LIN {X 0,Y 530.857,Z 807.028,A -85,B 0,C 180,E1 -4221.626,E2 -4221.626} C_VEL
LIN {X 0,Y 530.672,Z 814.477,A -85,B 0,C 180,E1 -4222.772,E2 -4222.772} C_VEL
LIN {X 0,Y 530.61,Z 820.462,A -85,B 0,C 180,E1 -4223.917,E2 -4223.917} C_VEL
LIN {X 0,Y 530.459,Z 825.2,A -85,B 0,C 180,E1 -4225.059,E2 -4225.059} C_VEL
LIN {X 0,Y 530.516,Z 828.828,A -85,B 0,C 180,E1 -4226.202,E2 -4226.202} C_VEL
LIN {X 0,Y 530.457,Z 830.697,A -85,B 0,C 180,E1 -4226.962,E2 -4226.962} C_VEL
LIN {X 0,Y 530.411,Z 832.131,A -85,B 0,C 180,E1 -4227.721,E2 -4227.721} C_VEL
LIN {X 0,Y 530.344,Z 833.756,A -85,B 0,C 180,E1 -4229.24,E2 -4229.24} C_VEL
LIN {X 0,Y 530.343,Z 833.996,A -85,B 0,C 180,E1 -4229.999,E2 -4229.999} C_VEL
LIN {X 0,Y 530.344,Z 833.813,A -85,B 0,C 180,E1 -4230.759,E2 -4230.759} C_VEL
LIN {X 0,Y 530.411,Z 832.265,A -85,B 0,C 180,E1 -4232.277,E2 -4232.277} C_VEL
LIN {X 0,Y 530.457,Z 830.904,A -85,B 0,C 180,E1 -4233.037,E2 -4233.037} C_VEL
LIN {X 0,Y 530.523,Z 828.033,A -85,B 0,C 180,E1 -4234.178,E2 -4234.178} C_VEL
LIN {X 0,Y 530.523,Z 824.133,A -85,B 0,C 180,E1 -4235.32,E2 -4235.32} C_VEL
LIN {X 0,Y 530.593,Z 818.515,A -85,B 0,C 180,E1 -4236.576,E2 -4236.576} C_VEL
LIN {X 0,Y 530.757,Z 811.537,A -85,B 0,C 180,E1 -4237.8,E2 -4237.8} C_VEL
LIN {X 0,Y 530.906,Z 803.362,A -85,B 0,C 180,E1 -4238.948,E2 -4238.948} C_VEL
LIN {X 0,Y 531.11,Z 794.95,A -85,B 0,C 180,E1 -4239.905,E2 -4239.905} C_VEL
LIN {X 0,Y 531.408,Z 784.646,A -85,B 0,C 180,E1 -4240.862,E2 -4240.862} C_VEL
LIN {X 0,Y 531.632,Z 773.907,A -85,B 0,C 180,E1 -4241.668,E2 -4241.668} C_VEL
LIN {X 0,Y 531.868,Z 763.248,A -85,B 0,C 180,E1 -4242.302,E2 -4242.302} C_VEL
LIN {X 0,Y 532.123,Z 750.651,A -85,B 0,C 180,E1 -4242.877,E2 -4242.877} C_VEL
LIN {X 0,Y 532.321,Z 738.262,A -85,B 0,C 180,E1 -4243.285,E2 -4243.285} C_VEL
LIN {X 0,Y 532.459,Z 725.504,A -85,B 0,C 180,E1 -4243.549,E2 -4243.549} C_VEL
LIN {X 0,Y 532.759,Z 629.988,A -85,B 0,C 180,E1 -4244.844,E2 -4244.844} C_VEL
LIN {X 0,Y 531.39,Z 621.592,A -85,B 0,C 180,E1 -4245.008,E2 -4245.008} C_VEL
LIN {X 0,Y 531.82,Z 600.643,A -85,B 0,C 180,E1 -4248.133,E2 -4248.133} C_VEL
LIN {X 0,Y 532.25,Z 580.755,A -85,B 0,C 180,E1 -4251.088,E2 -4251.088} C_VEL
LIN {X 0,Y 532.638,Z 561.67,A -85,B 0,C 180,E1 -4253.936,E2 -4253.936} C_VEL
LIN {X 0,Y 532.951,Z 545.283,A -85,B 0,C 180,E1 -4256.395,E2 -4256.395} C_VEL
LIN {X 0,Y 532.042,Z 539.407,A -85,B 0,C 180,E1 -4257.323,E2 -4257.323} C_VEL
LIN {X 0,Y 531.008,Z 534.341,A -85,B 0,C 180,E1 -4258.13,E2 -4258.13} C_VEL
LIN {X 0,Y 530.963,Z 534.35,A -85,B 0,C 180,E1 -4261.078,E2 -4261.078} C_VEL
LIN {X 0,Y 530.991,Z 534.342,A -85,B 0,C 180,E1 -4263.771,E2 -4263.771} C_VEL
LIN {X 0,Y 530.966,Z 534.341,A -85,B 0,C 180,E1 -4266.556,E2 -4266.556} C_VEL
LIN {X 0,Y 530.98,Z 534.341,A -85,B 0,C 180,E1 -4269.853,E2 -4269.853} C_VEL
LIN {X 0,Y 530.978,Z 534.339,A -85,B 0,C 180,E1 -4272.455,E2 -4272.455} C_VEL
LIN {X 0,Y 530.983,Z 534.344,A -85,B 0,C 180,E1 -4275.62,E2 -4275.62} C_VEL
LIN {X 0,Y 531.013,Z 534.336,A -85,B 0,C 180,E1 -4278.566,E2 -4278.566} C_VEL
LIN {X 0,Y 530.954,Z 534.351,A -85,B 0,C 180,E1 -4281.529,E2 -4281.529} C_VEL
LIN {X 0,Y 531.024,Z 534.342,A -85,B 0,C 180,E1 -4283.492,E2 -4283.492} C_VEL
LIN {X 0,Y 532.777,Z 540.518,A -85,B 0,C 180,E1 -4283.646,E2 -4283.646} C_VEL
LIN {X 0,Y 532.371,Z 613.502,A -85,B 0,C 180,E1 -4284.663,E2 -4284.663} C_VEL
LIN {X 0,Y 532.284,Z 626.553,A -85,B 0,C 180,E1 -4284.993,E2 -4284.993} C_VEL
LIN {X 0,Y 532.14,Z 640.049,A -85,B 0,C 180,E1 -4285.51,E2 -4285.51} C_VEL
LIN {X 0,Y 531.967,Z 650.777,A -85,B 0,C 180,E1 -4286.07,E2 -4286.07} C_VEL
LIN {X 0,Y 531.745,Z 660.944,A -85,B 0,C 180,E1 -4286.736,E2 -4286.736} C_VEL
LIN {X 0,Y 531.534,Z 670.886,A -85,B 0,C 180,E1 -4287.54,E2 -4287.54} C_VEL
LIN {X 0,Y 531.32,Z 680.523,A -85,B 0,C 180,E1 -4288.501,E2 -4288.501} C_VEL
LIN {X 0,Y 531.11,Z 689.206,A -85,B 0,C 180,E1 -4289.568,E2 -4289.568} C_VEL
LIN {X 0,Y 530.906,Z 696.438,A -85,B 0,C 180,E1 -4290.673,E2 -4290.673} C_VEL
LIN {X 0,Y 530.761,Z 703.132,A -85,B 0,C 180,E1 -4291.961,E2 -4291.961} C_VEL
LIN {X 0,Y 530.695,Z 708.251,A -85,B 0,C 180,E1 -4293.239,E2 -4293.239} C_VEL
LIN {X 0,Y 530.658,Z 711.26,A -85,B 0,C 180,E1 -4294.232,E2 -4294.232} C_VEL
LIN {X 0,Y 530.576,Z 712.968,A -85,B 0,C 180,E1 -4294.921,E2 -4294.921} C_VEL
LIN {X 0,Y 530.54,Z 714.979,A -85,B 0,C 180,E1 -4296.065,E2 -4296.065} C_VEL
LIN {X 0,Y 530.53,Z 716.161,A -85,B 0,C 180,E1 -4297.408,E2 -4297.408} C_VEL
LIN {X 0,Y 530.522,Z 716.323,A -85,B 0,C 180,E1 -4298.227,E2 -4298.227} C_VEL
LIN {X 0,Y 530.549,Z 716.011,A -85,B 0,C 180,E1 -4299.043,E2 -4299.043} C_VEL
LIN {X 0,Y 530.546,Z 714.9,A -85,B 0,C 180,E1 -4300.134,E2 -4300.134} C_VEL
LIN {X 0,Y 530.626,Z 712.421,A -85,B 0,C 180,E1 -4301.466,E2 -4301.466} C_VEL
LIN {X 0,Y 530.723,Z 708.756,A -85,B 0,C 180,E1 -4302.759,E2 -4302.759} C_VEL
LIN {X 0,Y 530.787,Z 704.588,A -85,B 0,C 180,E1 -4303.856,E2 -4303.856} C_VEL
LIN {X 0,Y 530.918,Z 698.585,A -85,B 0,C 180,E1 -4305.085,E2 -4305.085} C_VEL
LIN {X 0,Y 531.091,Z 691.628,A -85,B 0,C 180,E1 -4306.22,E2 -4306.22} C_VEL
LIN {X 0,Y 531.32,Z 682.636,A -85,B 0,C 180,E1 -4307.393,E2 -4307.393} C_VEL
LIN {X 0,Y 531.545,Z 672.652,A -85,B 0,C 180,E1 -4308.427,E2 -4308.427} C_VEL
LIN {X 0,Y 531.81,Z 662.883,A -85,B 0,C 180,E1 -4309.242,E2 -4309.242} C_VEL
LIN {X 0,Y 531.97,Z 652.92,A -85,B 0,C 180,E1 -4309.918,E2 -4309.918} C_VEL
LIN {X 0,Y 532.165,Z 641.21,A -85,B 0,C 180,E1 -4310.546,E2 -4310.546} C_VEL
LIN {X 0,Y 532.316,Z 628.322,A -85,B 0,C 180,E1 -4311.052,E2 -4311.052} C_VEL
LIN {X 0,Y 532.423,Z 615.599,A -85,B 0,C 180,E1 -4311.388,E2 -4311.388} C_VEL
LIN {X 0,Y 532.528,Z 579.636,A -85,B 0,C 180,E1 -4311.911,E2 -4311.911} C_VEL
LIN {X 0,Y 532.662,Z 539.432,A -85,B 0,C 180,E1 -4312.471,E2 -4312.471} C_VEL
LIN {X 0,Y 531.058,Z 534.338,A -85,B 0,C 180,E1 -4312.605,E2 -4312.605} C_VEL
LIN {X 0,Y 531.137,Z 534.329,A -85,B 0,C 180,E1 -4314.685,E2 -4314.685} C_VEL
LIN {X 0,Y 531.13,Z 534.321,A -85,B 0,C 180,E1 -4317.725,E2 -4317.725} C_VEL
LIN {X 0,Y 531.147,Z 534.328,A -85,B 0,C 180,E1 -4320.758,E2 -4320.758} C_VEL
LIN {X 0,Y 531.101,Z 534.329,A -85,B 0,C 180,E1 -4323.034,E2 -4323.034} C_VEL
LIN {X 0,Y 531.081,Z 534.328,A -85,B 0,C 180,E1 -4326.077,E2 -4326.077} C_VEL
LIN {X 0,Y 531.027,Z 534.336,A -85,B 0,C 180,E1 -4329.138,E2 -4329.138} C_VEL
LIN {X 0,Y 531.03,Z 534.335,A -85,B 0,C 180,E1 -4332.225,E2 -4332.225} C_VEL
LIN {X 0,Y 530.985,Z 534.338,A -85,B 0,C 180,E1 -4335.35,E2 -4335.35} C_VEL
LIN {X 0,Y 531.006,Z 534.336,A -85,B 0,C 180,E1 -4337.723,E2 -4337.723} C_VEL
LIN {X 0,Y 530.992,Z 534.344,A -85,B 0,C 180,E1 -4340.938,E2 -4340.938} C_VEL
LIN {X 0,Y 530.97,Z 534.342,A -85,B 0,C 180,E1 -4344.225,E2 -4344.225} C_VEL
LIN {X 0,Y 531.003,Z 534.344,A -85,B 0,C 180,E1 -4346.744,E2 -4346.744} C_VEL
LIN {X 0,Y 530.991,Z 534.34,A -85,B 0,C 180,E1 -4349.322,E2 -4349.322} C_VEL
LIN {X 0,Y 530.972,Z 534.341,A -85,B 0,C 180,E1 -4352.104,E2 -4352.104} C_VEL
LIN {X 0,Y 530.984,Z 534.345,A -85,B 0,C 180,E1 -4354.856,E2 -4354.856} C_VEL
LIN {X 0,Y 530.96,Z 534.341,A -85,B 0,C 180,E1 -4357.508,E2 -4357.508} C_VEL
LIN {X 0,Y 531.021,Z 534.337,A -85,B 0,C 180,E1 -4360.429,E2 -4360.429} C_VEL
LIN {X 0,Y 530.962,Z 534.344,A -85,B 0,C 180,E1 -4363.495,E2 -4363.495} C_VEL
LIN {X 0,Y 530.961,Z 534.347,A -85,B 0,C 180,E1 -4366.507,E2 -4366.507} C_VEL
LIN {X 0,Y 531.004,Z 534.338,A -85,B 0,C 180,E1 -4369.571,E2 -4369.571} C_VEL
LIN {X 0,Y 530.974,Z 534.346,A -85,B 0,C 180,E1 -4372.577,E2 -4372.577} C_VEL
LIN {X 0,Y 531.001,Z 534.341,A -85,B 0,C 180,E1 -4375.312,E2 -4375.312} C_VEL
LIN {X 0,Y 530.981,Z 534.341,A -85,B 0,C 180,E1 -4378.034,E2 -4378.034} C_VEL
LIN {X 0,Y 530.988,Z 534.347,A -85,B 0,C 180,E1 -4380.875,E2 -4380.875} C_VEL
LIN {X 0,Y 531.045,Z 534.42,A -85,B 0,C 180,E1 -4381.672,E2 -4381.672} C_VEL
LIN {X 0,Y 533.486,Z 546.142,A -85,B 0,C 180,E1 -4383.18,E2 -4383.18} C_VEL
LIN {X 0,Y 533.098,Z 569.291,A -85,B 0,C 180,E1 -4385.879,E2 -4385.879} C_VEL
LIN {X 0,Y 532.644,Z 593.969,A -85,B 0,C 180,E1 -4388.726,E2 -4388.726} C_VEL
LIN {X 0,Y 532.2,Z 621.201,A -85,B 0,C 180,E1 -4391.799,E2 -4391.799} C_VEL
LIN {X 0,Y 531.716,Z 649.824,A -85,B 0,C 180,E1 -4395.024,E2 -4395.024} C_VEL
LIN {X 0,Y 532.846,Z 659.307,A -85,B 0,C 180,E1 -4395.194,E2 -4395.194} C_VEL
LIN {X 0,Y 532.428,Z 759.985,A -85,B 0,C 180,E1 -4396.572,E2 -4396.572} C_VEL
LIN {X 0,Y 532.25,Z 773.234,A -85,B 0,C 180,E1 -4396.908,E2 -4396.908} C_VEL
LIN {X 0,Y 532.06,Z 785.381,A -85,B 0,C 180,E1 -4397.364,E2 -4397.364} C_VEL
LIN {X 0,Y 531.805,Z 797.318,A -85,B 0,C 180,E1 -4397.968,E2 -4397.968} C_VEL
LIN {X 0,Y 531.534,Z 809.205,A -85,B 0,C 180,E1 -4398.755,E2 -4398.755} C_VEL
LIN {X 0,Y 531.255,Z 819.613,A -85,B 0,C 180,E1 -4399.617,E2 -4399.617} C_VEL
LIN {X 0,Y 531.06,Z 828.121,A -85,B 0,C 180,E1 -4400.479,E2 -4400.479} C_VEL
LIN {X 0,Y 530.886,Z 835.966,A -85,B 0,C 180,E1 -4401.436,E2 -4401.436} C_VEL
LIN {X 0,Y 530.684,Z 843.627,A -85,B 0,C 180,E1 -4402.582,E2 -4402.582} C_VEL
LIN {X 0,Y 530.604,Z 850.682,A -85,B 0,C 180,E1 -4403.918,E2 -4403.918} C_VEL
LIN {X 0,Y 530.459,Z 855.375,A -85,B 0,C 180,E1 -4405.06,E2 -4405.06} C_VEL
LIN {X 0,Y 530.516,Z 858.962,A -85,B 0,C 180,E1 -4406.203,E2 -4406.203} C_VEL
LIN {X 0,Y 530.457,Z 860.811,A -85,B 0,C 180,E1 -4406.963,E2 -4406.963} C_VEL
LIN {X 0,Y 530.41,Z 862.198,A -85,B 0,C 180,E1 -4407.723,E2 -4407.723} C_VEL
LIN {X 0,Y 530.344,Z 863.787,A -85,B 0,C 180,E1 -4409.241,E2 -4409.241} C_VEL
LIN {X 0,Y 530.342,Z 864,A -85,B 0,C 180,E1 -4410.001,E2 -4410.001} C_VEL
LIN {X 0,Y 530.361,Z 863.182,A -85,B 0,C 180,E1 -4411.519,E2 -4411.519} C_VEL
LIN {X 0,Y 530.41,Z 862.193,A -85,B 0,C 180,E1 -4412.279,E2 -4412.279} C_VEL
LIN {X 0,Y 530.457,Z 860.806,A -85,B 0,C 180,E1 -4413.038,E2 -4413.038} C_VEL
LIN {X 0,Y 530.523,Z 857.893,A -85,B 0,C 180,E1 -4414.179,E2 -4414.179} C_VEL
LIN {X 0,Y 530.525,Z 853.948,A -85,B 0,C 180,E1 -4415.321,E2 -4415.321} C_VEL
LIN {X 0,Y 530.599,Z 848.261,A -85,B 0,C 180,E1 -4416.582,E2 -4416.582} C_VEL
LIN {X 0,Y 530.759,Z 841.232,A -85,B 0,C 180,E1 -4417.801,E2 -4417.801} C_VEL
LIN {X 0,Y 530.93,Z 832.988,A -85,B 0,C 180,E1 -4418.948,E2 -4418.948} C_VEL
LIN {X 0,Y 531.137,Z 824.535,A -85,B 0,C 180,E1 -4419.906,E2 -4419.906} C_VEL
LIN {X 0,Y 531.409,Z 814.086,A -85,B 0,C 180,E1 -4420.863,E2 -4420.863} C_VEL
LIN {X 0,Y 531.694,Z 803.348,A -85,B 0,C 180,E1 -4421.656,E2 -4421.656} C_VEL
LIN {X 0,Y 531.933,Z 792.398,A -85,B 0,C 180,E1 -4422.301,E2 -4422.301} C_VEL
LIN {X 0,Y 532.145,Z 780.762,A -85,B 0,C 180,E1 -4422.829,E2 -4422.829} C_VEL
LIN {X 0,Y 532.302,Z 767.334,A -85,B 0,C 180,E1 -4423.262,E2 -4423.262} C_VEL
LIN {X 0,Y 532.481,Z 754.055,A -85,B 0,C 180,E1 -4423.525,E2 -4423.525} C_VEL
LIN {X 0,Y 532.704,Z 658.004,A -85,B 0,C 180,E1 -4424.828,E2 -4424.828} C_VEL
LIN {X 0,Y 531.593,Z 650.618,A -85,B 0,C 180,E1 -4424.969,E2 -4424.969} C_VEL
LIN {X 0,Y 531.951,Z 627.9,A -85,B 0,C 180,E1 -4427.853,E2 -4427.853} C_VEL
LIN {X 0,Y 532.42,Z 604.132,A -85,B 0,C 180,E1 -4430.88,E2 -4430.88} C_VEL
LIN {X 0,Y 532.824,Z 580.756,A -85,B 0,C 180,E1 -4433.929,E2 -4433.929} C_VEL
LIN {X 0,Y 533.285,Z 560.404,A -85,B 0,C 180,E1 -4436.621,E2 -4436.621} C_VEL
LIN {X 0,Y 533.55,Z 546.301,A -85,B 0,C 180,E1 -4438.522,E2 -4438.522} C_VEL
LIN {X 0,Y 530.999,Z 534.344,A -85,B 0,C 180,E1 -4440.312,E2 -4440.312} C_VEL
LIN {X 0,Y 531.002,Z 534.34,A -85,B 0,C 180,E1 -4443.506,E2 -4443.506} C_VEL
LIN {X 0,Y 530.958,Z 534.345,A -85,B 0,C 180,E1 -4446.558,E2 -4446.558} C_VEL
LIN {X 0,Y 530.991,Z 534.341,A -85,B 0,C 180,E1 -4449.443,E2 -4449.443} C_VEL
LIN {X 0,Y 530.98,Z 534.34,A -85,B 0,C 180,E1 -4452.457,E2 -4452.457} C_VEL
LIN {X 0,Y 530.99,Z 534.34,A -85,B 0,C 180,E1 -4455.621,E2 -4455.621} C_VEL
LIN {X 0,Y 531.002,Z 534.334,A -85,B 0,C 180,E1 -4458.565,E2 -4458.565} C_VEL
LIN {X 0,Y 530.961,Z 534.344,A -85,B 0,C 180,E1 -4461.529,E2 -4461.529} C_VEL
LIN {X 0,Y 530.983,Z 534.336,A -85,B 0,C 180,E1 -4464.382,E2 -4464.382} C_VEL
LIN {X 0,Y 530.971,Z 534.347,A -85,B 0,C 180,E1 -4467.134,E2 -4467.134} C_VEL
LIN {X 0,Y 530.97,Z 534.341,A -85,B 0,C 180,E1 -4469.803,E2 -4469.803} C_VEL
LIN {X 0,Y 531.015,Z 534.334,A -85,B 0,C 180,E1 -4472.467,E2 -4472.467} C_VEL
LIN {X 0,Y 531.005,Z 534.336,A -85,B 0,C 180,E1 -4474.942,E2 -4474.942} C_VEL
LIN {X 0,Y 530.971,Z 534.34,A -85,B 0,C 180,E1 -4478.247,E2 -4478.247} C_VEL
LIN {X 0,Y 530.995,Z 534.335,A -85,B 0,C 180,E1 -4480.677,E2 -4480.677} C_VEL
LIN {X 0,Y 530.986,Z 534.335,A -85,B 0,C 180,E1 -4483.071,E2 -4483.071} C_VEL
LIN {X 0,Y 531.04,Z 534.339,A -85,B 0,C 180,E1 -4485.436,E2 -4485.436} C_VEL
LIN {X 0,Y 531.036,Z 534.327,A -85,B 0,C 180,E1 -4488.55,E2 -4488.55} C_VEL
LIN {X 0,Y 531.056,Z 534.336,A -85,B 0,C 180,E1 -4491.629,E2 -4491.629} C_VEL
LIN {X 0,Y 531.121,Z 534.32,A -85,B 0,C 180,E1 -4494.685,E2 -4494.685} C_VEL
LIN {X 0,Y 531.139,Z 534.321,A -85,B 0,C 180,E1 -4497.725,E2 -4497.725} C_VEL
LIN {X 0,Y 531.153,Z 534.317,A -85,B 0,C 180,E1 -4500.758,E2 -4500.758} C_VEL
LIN {X 0,Y 531.107,Z 534.322,A -85,B 0,C 180,E1 -4503.034,E2 -4503.034} C_VEL
LIN {X 0,Y 531.083,Z 534.328,A -85,B 0,C 180,E1 -4506.077,E2 -4506.077} C_VEL
LIN {X 0,Y 531.031,Z 534.333,A -85,B 0,C 180,E1 -4509.138,E2 -4509.138} C_VEL
LIN {X 0,Y 531.04,Z 534.329,A -85,B 0,C 180,E1 -4512.225,E2 -4512.225} C_VEL
LIN {X 0,Y 530.995,Z 534.338,A -85,B 0,C 180,E1 -4515.35,E2 -4515.35} C_VEL
LIN {X 0,Y 530.992,Z 534.334,A -85,B 0,C 180,E1 -4518.521,E2 -4518.521} C_VEL
LIN {X 0,Y 531,Z 534.335,A -85,B 0,C 180,E1 -4520.938,E2 -4520.938} C_VEL
LIN {X 0,Y 530.98,Z 534.341,A -85,B 0,C 180,E1 -4524.225,E2 -4524.225} C_VEL
LIN {X 0,Y 531.004,Z 534.335,A -85,B 0,C 180,E1 -4526.744,E2 -4526.744} C_VEL
LIN {X 0,Y 530.982,Z 534.339,A -85,B 0,C 180,E1 -4529.323,E2 -4529.323} C_VEL
LIN {X 0,Y 530.966,Z 534.348,A -85,B 0,C 180,E1 -4532.1,E2 -4532.1} C_VEL
LIN {X 0,Y 530.971,Z 534.339,A -85,B 0,C 180,E1 -4534.851,E2 -4534.851} C_VEL
LIN {X 0,Y 530.967,Z 534.342,A -85,B 0,C 180,E1 -4537.508,E2 -4537.508} C_VEL
LIN {X 0,Y 530.986,Z 534.345,A -85,B 0,C 180,E1 -4540.433,E2 -4540.433} C_VEL
LIN {X 0,Y 530.968,Z 534.338,A -85,B 0,C 180,E1 -4543.282,E2 -4543.282} C_VEL
LIN {X 0,Y 530.963,Z 534.34,A -85,B 0,C 180,E1 -4543.567,E2 -4543.567} C_VEL
LIN {X 0,Y 530.285,Z 534.433,A -85,B 0,C 180,E1 -4544.201,E2 -4544.201} C_VEL
LIN {X 0,Y 527.427,Z 534.783,A -85,B 0,C 180,E1 -4545.229,E2 -4545.229} C_VEL
LIN {X 0,Y 525.019,Z 535.088,A -85,B 0,C 180,E1 -4546.057,E2 -4546.057} C_VEL
LIN {X 0,Y 523.989,Z 535.207,A -85,B 0,C 180,E1 -4546.697,E2 -4546.697} C_VEL
LIN {X 0,Y 523.907,Z 535.215,A -85,B 0,C 180,E1 -4546.914,E2 -4546.914} C_VEL
LIN {X 0,Y 523.951,Z 535.219,A -85,B 0,C 180,E1 -4549.921,E2 -4549.921} C_VEL
LIN {X 0,Y 523.911,Z 535.222,A -85,B 0,C 180,E1 -4552.868,E2 -4552.868} C_VEL
LIN {X 0,Y 523.944,Z 535.218,A -85,B 0,C 180,E1 -4555.71,E2 -4555.71} C_VEL
LIN {X 0,Y 523.927,Z 535.226,A -85,B 0,C 180,E1 -4558.456,E2 -4558.456} C_VEL
LIN {X 0,Y 523.943,Z 535.22,A -85,B 0,C 180,E1 -4561.125,E2 -4561.125} C_VEL
LIN {X 0,Y 523.977,Z 535.252,A -85,B 0,C 180,E1 -4563.272,E2 -4563.272} C_VEL
LIN {X 0,Y 526.189,Z 546.301,A -85,B 0,C 180,E1 -4564.868,E2 -4564.868} C_VEL
LIN {X 0,Y 525.813,Z 563.993,A -85,B 0,C 180,E1 -4567.258,E2 -4567.258} C_VEL
LIN {X 0,Y 525.367,Z 586.308,A -85,B 0,C 180,E1 -4570.258,E2 -4570.258} C_VEL
LIN {X 0,Y 524.854,Z 607.393,A -85,B 0,C 180,E1 -4573.067,E2 -4573.067} C_VEL
LIN {X 0,Y 524.574,Z 620.937,A -85,B 0,C 180,E1 -4574.882,E2 -4574.882} C_VEL
LIN {X 0,Y 525.951,Z 631.321,A -85,B 0,C 180,E1 -4575.068,E2 -4575.068} C_VEL
LIN {X 0,Y 525.592,Z 730.102,A -85,B 0,C 180,E1 -4576.442,E2 -4576.442} C_VEL
LIN {X 0,Y 525.351,Z 742.698,A -85,B 0,C 180,E1 -4576.756,E2 -4576.756} C_VEL
LIN {X 0,Y 525.075,Z 755.532,A -85,B 0,C 180,E1 -4577.241,E2 -4577.241} C_VEL
LIN {X 0,Y 524.813,Z 768.516,A -85,B 0,C 180,E1 -4577.919,E2 -4577.919} C_VEL
LIN {X 0,Y 524.579,Z 779.937,A -85,B 0,C 180,E1 -4578.7,E2 -4578.7} C_VEL
LIN {X 0,Y 524.238,Z 790.15,A -85,B 0,C 180,E1 -4579.573,E2 -4579.573} C_VEL
LIN {X 0,Y 523.99,Z 799.413,A -85,B 0,C 180,E1 -4580.543,E2 -4580.543} C_VEL
LIN {X 0,Y 523.769,Z 808.366,A -85,B 0,C 180,E1 -4581.706,E2 -4581.706} C_VEL
LIN {X 0,Y 523.588,Z 815.567,A -85,B 0,C 180,E1 -4582.867,E2 -4582.867} C_VEL
LIN {X 0,Y 523.546,Z 822.19,A -85,B 0,C 180,E1 -4584.221,E2 -4584.221} C_VEL
LIN {X 0,Y 523.361,Z 826.54,A -85,B 0,C 180,E1 -4585.378,E2 -4585.378} C_VEL
LIN {X 0,Y 523.444,Z 828.829,A -85,B 0,C 180,E1 -4586.15,E2 -4586.15} C_VEL
LIN {X 0,Y 523.368,Z 830.698,A -85,B 0,C 180,E1 -4586.92,E2 -4586.92} C_VEL
LIN {X 0,Y 523.335,Z 832.132,A -85,B 0,C 180,E1 -4587.69,E2 -4587.69} C_VEL
LIN {X 0,Y 523.25,Z 833.756,A -85,B 0,C 180,E1 -4589.23,E2 -4589.23} C_VEL
LIN {X 0,Y 523.247,Z 833.997,A -85,B 0,C 180,E1 -4589.999,E2 -4589.999} C_VEL
LIN {X 0,Y 523.25,Z 833.812,A -85,B 0,C 180,E1 -4590.769,E2 -4590.769} C_VEL
LIN {X 0,Y 523.335,Z 832.264,A -85,B 0,C 180,E1 -4592.308,E2 -4592.308} C_VEL
LIN {X 0,Y 523.368,Z 830.902,A -85,B 0,C 180,E1 -4593.078,E2 -4593.078} C_VEL
LIN {X 0,Y 523.442,Z 828.031,A -85,B 0,C 180,E1 -4594.234,E2 -4594.234} C_VEL
LIN {X 0,Y 523.463,Z 824.131,A -85,B 0,C 180,E1 -4595.392,E2 -4595.392} C_VEL
LIN {X 0,Y 523.517,Z 818.972,A -85,B 0,C 180,E1 -4596.574,E2 -4596.574} C_VEL
LIN {X 0,Y 523.687,Z 811.531,A -85,B 0,C 180,E1 -4597.906,E2 -4597.906} C_VEL
LIN {X 0,Y 523.875,Z 803.356,A -85,B 0,C 180,E1 -4599.069,E2 -4599.069} C_VEL
LIN {X 0,Y 524.092,Z 794.941,A -85,B 0,C 180,E1 -4600.039,E2 -4600.039} C_VEL
LIN {X 0,Y 524.435,Z 784.667,A -85,B 0,C 180,E1 -4601.008,E2 -4601.008} C_VEL
LIN {X 0,Y 524.662,Z 774.366,A -85,B 0,C 180,E1 -4601.797,E2 -4601.797} C_VEL
LIN {X 0,Y 524.936,Z 763.313,A -85,B 0,C 180,E1 -4602.467,E2 -4602.467} C_VEL
LIN {X 0,Y 525.205,Z 750.727,A -85,B 0,C 180,E1 -4603.05,E2 -4603.05} C_VEL
LIN {X 0,Y 525.432,Z 738.334,A -85,B 0,C 180,E1 -4603.462,E2 -4603.462} C_VEL
LIN {X 0,Y 525.576,Z 725.581,A -85,B 0,C 180,E1 -4603.729,E2 -4603.729} C_VEL
LIN {X 0,Y 525.86,Z 630.572,A -85,B 0,C 180,E1 -4605.035,E2 -4605.035} C_VEL
LIN {X 0,Y 524.424,Z 621.641,A -85,B 0,C 180,E1 -4605.211,E2 -4605.211} C_VEL
LIN {X 0,Y 524.861,Z 601.08,A -85,B 0,C 180,E1 -4608.299,E2 -4608.299} C_VEL
LIN {X 0,Y 525.284,Z 581.86,A -85,B 0,C 180,E1 -4611.176,E2 -4611.176} C_VEL
LIN {X 0,Y 525.723,Z 562.71,A -85,B 0,C 180,E1 -4614.061,E2 -4614.061} C_VEL
LIN {X 0,Y 526.014,Z 545.667,A -85,B 0,C 180,E1 -4616.656,E2 -4616.656} C_VEL
LIN {X 0,Y 523.972,Z 535.219,A -85,B 0,C 180,E1 -4618.352,E2 -4618.352} C_VEL
LIN {X 0,Y 523.93,Z 535.223,A -85,B 0,C 180,E1 -4621.542,E2 -4621.542} C_VEL
LIN {X 0,Y 523.944,Z 535.218,A -85,B 0,C 180,E1 -4624.288,E2 -4624.288} C_VEL
LIN {X 0,Y 523.913,Z 535.226,A -85,B 0,C 180,E1 -4627.13,E2 -4627.13} C_VEL
LIN {X 0,Y 523.932,Z 535.217,A -85,B 0,C 180,E1 -4630.129,E2 -4630.129} C_VEL
LIN {X 0,Y 523.935,Z 535.216,A -85,B 0,C 180,E1 -4632.458,E2 -4632.458} C_VEL
LIN {X 0,Y 523.951,Z 535.221,A -85,B 0,C 180,E1 -4635.307,E2 -4635.307} C_VEL
LIN {X 0,Y 523.976,Z 535.213,A -85,B 0,C 180,E1 -4638.685,E2 -4638.685} C_VEL
LIN {X 0,Y 523.947,Z 535.221,A -85,B 0,C 180,E1 -4641.074,E2 -4641.074} C_VEL
LIN {X 0,Y 523.976,Z 535.268,A -85,B 0,C 180,E1 -4643.313,E2 -4643.313} C_VEL
LIN {X 0,Y 525.906,Z 541.232,A -85,B 0,C 180,E1 -4643.456,E2 -4643.456} C_VEL
LIN {X 0,Y 525.522,Z 614.868,A -85,B 0,C 180,E1 -4644.506,E2 -4644.506} C_VEL
LIN {X 0,Y 525.411,Z 628.218,A -85,B 0,C 180,E1 -4644.857,E2 -4644.857} C_VEL
LIN {X 0,Y 525.266,Z 640.719,A -85,B 0,C 180,E1 -4645.344,E2 -4645.344} C_VEL
LIN {X 0,Y 525.076,Z 651.455,A -85,B 0,C 180,E1 -4645.905,E2 -4645.905} C_VEL
LIN {X 0,Y 524.825,Z 662.003,A -85,B 0,C 180,E1 -4646.604,E2 -4646.604} C_VEL
LIN {X 0,Y 524.575,Z 672.723,A -85,B 0,C 180,E1 -4647.493,E2 -4647.493} C_VEL
LIN {X 0,Y 524.336,Z 682.377,A -85,B 0,C 180,E1 -4648.483,E2 -4648.483} C_VEL
LIN {X 0,Y 524.124,Z 691.021,A -85,B 0,C 180,E1 -4649.589,E2 -4649.589} C_VEL
LIN {X 0,Y 523.902,Z 697.976,A -85,B 0,C 180,E1 -4650.684,E2 -4650.684} C_VEL
LIN {X 0,Y 523.762,Z 704.572,A -85,B 0,C 180,E1 -4651.989,E2 -4651.989} C_VEL
LIN {X 0,Y 523.71,Z 709.592,A -85,B 0,C 180,E1 -4653.284,E2 -4653.284} C_VEL
LIN {X 0,Y 523.593,Z 713.226,A -85,B 0,C 180,E1 -4654.562,E2 -4654.562} C_VEL
LIN {X 0,Y 523.537,Z 715.764,A -85,B 0,C 180,E1 -4655.897,E2 -4655.897} C_VEL
LIN {X 0,Y 523.498,Z 717.012,A -85,B 0,C 180,E1 -4657.087,E2 -4657.087} C_VEL
LIN {X 0,Y 523.514,Z 717.334,A -85,B 0,C 180,E1 -4657.92,E2 -4657.92} C_VEL
LIN {X 0,Y 523.531,Z 717.191,A -85,B 0,C 180,E1 -4658.749,E2 -4658.749} C_VEL
LIN {X 0,Y 523.53,Z 716.142,A -85,B 0,C 180,E1 -4659.996,E2 -4659.996} C_VEL
LIN {X 0,Y 523.599,Z 714.112,A -85,B 0,C 180,E1 -4661.207,E2 -4661.207} C_VEL
LIN {X 0,Y 523.671,Z 711.297,A -85,B 0,C 180,E1 -4662.333,E2 -4662.333} C_VEL
LIN {X 0,Y 523.763,Z 706.82,A -85,B 0,C 180,E1 -4663.633,E2 -4663.633} C_VEL
LIN {X 0,Y 523.942,Z 700.744,A -85,B 0,C 180,E1 -4664.963,E2 -4664.963} C_VEL
LIN {X 0,Y 524.106,Z 694.572,A -85,B 0,C 180,E1 -4666.032,E2 -4666.032} C_VEL
LIN {X 0,Y 524.285,Z 687.599,A -85,B 0,C 180,E1 -4667.025,E2 -4667.025} C_VEL
LIN {X 0,Y 524.495,Z 679.311,A -85,B 0,C 180,E1 -4667.998,E2 -4667.998} C_VEL
LIN {X 0,Y 524.728,Z 668.738,A -85,B 0,C 180,E1 -4668.997,E2 -4668.997} C_VEL
LIN {X 0,Y 525.001,Z 658.347,A -85,B 0,C 180,E1 -4669.783,E2 -4669.783} C_VEL
LIN {X 0,Y 525.253,Z 646.898,A -85,B 0,C 180,E1 -4670.469,E2 -4670.469} C_VEL
LIN {X 0,Y 525.386,Z 635.089,A -85,B 0,C 180,E1 -4671.005,E2 -4671.005} C_VEL
LIN {X 0,Y 525.47,Z 621.492,A -85,B 0,C 180,E1 -4671.443,E2 -4671.443} C_VEL
LIN {X 0,Y 525.532,Z 607.858,A -85,B 0,C 180,E1 -4671.703,E2 -4671.703} C_VEL
LIN {X 0,Y 525.865,Z 540.993,A -85,B 0,C 180,E1 -4672.645,E2 -4672.645} C_VEL
LIN {X 0,Y 524.031,Z 535.214,A -85,B 0,C 180,E1 -4672.787,E2 -4672.787} C_VEL
LIN {X 0,Y 524.094,Z 535.206,A -85,B 0,C 180,E1 -4674.614,E2 -4674.614} C_VEL
LIN {X 0,Y 524.102,Z 535.197,A -85,B 0,C 180,E1 -4677.694,E2 -4677.694} C_VEL
LIN {X 0,Y 524.117,Z 535.203,A -85,B 0,C 180,E1 -4680.768,E2 -4680.768} C_VEL
LIN {X 0,Y 524.068,Z 535.204,A -85,B 0,C 180,E1 -4683.075,E2 -4683.075} C_VEL
LIN {X 0,Y 524.041,Z 535.205,A -85,B 0,C 180,E1 -4686.159,E2 -4686.159} C_VEL
LIN {X 0,Y 523.994,Z 535.211,A -85,B 0,C 180,E1 -4689.262,E2 -4689.262} C_VEL
LIN {X 0,Y 524.013,Z 535.207,A -85,B 0,C 180,E1 -4691.752,E2 -4691.752} C_VEL
LIN {X 0,Y 523.982,Z 535.213,A -85,B 0,C 180,E1 -4695.053,E2 -4695.053} C_VEL
LIN {X 0,Y 523.954,Z 535.215,A -85,B 0,C 180,E1 -4697.969,E2 -4697.969} C_VEL
LIN {X 0,Y 523.962,Z 535.217,A -85,B 0,C 180,E1 -4700.41,E2 -4700.41} C_VEL
LIN {X 0,Y 523.907,Z 535.228,A -85,B 0,C 180,E1 -4702.894,E2 -4702.894} C_VEL
LIN {X 0,Y 523.945,Z 535.216,A -85,B 0,C 180,E1 -4705.419,E2 -4705.419} C_VEL
LIN {X 0,Y 523.962,Z 535.213,A -85,B 0,C 180,E1 -4707.999,E2 -4707.999} C_VEL
LIN {X 0,Y 523.944,Z 535.224,A -85,B 0,C 180,E1 -4710.857,E2 -4710.857} C_VEL
LIN {X 0,Y 523.955,Z 535.214,A -85,B 0,C 180,E1 -4713.736,E2 -4713.736} C_VEL
LIN {X 0,Y 523.918,Z 535.223,A -85,B 0,C 180,E1 -4716.406,E2 -4716.406} C_VEL
LIN {X 0,Y 523.953,Z 535.22,A -85,B 0,C 180,E1 -4719.082,E2 -4719.082} C_VEL
LIN {X 0,Y 523.96,Z 535.215,A -85,B 0,C 180,E1 -4722.118,E2 -4722.118} C_VEL
LIN {X 0,Y 523.95,Z 535.219,A -85,B 0,C 180,E1 -4725.31,E2 -4725.31} C_VEL
LIN {X 0,Y 523.968,Z 535.22,A -85,B 0,C 180,E1 -4728.689,E2 -4728.689} C_VEL
LIN {X 0,Y 523.949,Z 535.222,A -85,B 0,C 180,E1 -4731.077,E2 -4731.077} C_VEL
LIN {X 0,Y 523.927,Z 535.22,A -85,B 0,C 180,E1 -4733.829,E2 -4733.829} C_VEL
LIN {X 0,Y 523.942,Z 535.223,A -85,B 0,C 180,E1 -4736.637,E2 -4736.637} C_VEL
LIN {X 0,Y 523.954,Z 535.221,A -85,B 0,C 180,E1 -4739.357,E2 -4739.357} C_VEL
LIN {X 0,Y 523.99,Z 535.296,A -85,B 0,C 180,E1 -4741.485,E2 -4741.485} C_VEL
LIN {X 0,Y 526.593,Z 547.998,A -85,B 0,C 180,E1 -4743.143,E2 -4743.143} C_VEL
LIN {X 0,Y 526.137,Z 571.739,A -85,B 0,C 180,E1 -4745.959,E2 -4745.959} C_VEL
LIN {X 0,Y 525.578,Z 598.018,A -85,B 0,C 180,E1 -4749.026,E2 -4749.026} C_VEL
LIN {X 0,Y 525.073,Z 624.677,A -85,B 0,C 180,E1 -4752.071,E2 -4752.071} C_VEL
LIN {X 0,Y 524.67,Z 649.011,A -85,B 0,C 180,E1 -4754.83,E2 -4754.83} C_VEL
LIN {X 0,Y 525.959,Z 659.644,A -85,B 0,C 180,E1 -4755.016,E2 -4755.016} C_VEL
LIN {X 0,Y 525.515,Z 759.406,A -85,B 0,C 180,E1 -4756.392,E2 -4756.392} C_VEL
LIN {X 0,Y 525.324,Z 772.875,A -85,B 0,C 180,E1 -4756.732,E2 -4756.732} C_VEL
LIN {X 0,Y 525.127,Z 785.226,A -85,B 0,C 180,E1 -4757.194,E2 -4757.194} C_VEL
LIN {X 0,Y 524.879,Z 796.026,A -85,B 0,C 180,E1 -4757.734,E2 -4757.734} C_VEL
LIN {X 0,Y 524.632,Z 806.604,A -85,B 0,C 180,E1 -4758.409,E2 -4758.409} C_VEL
LIN {X 0,Y 524.329,Z 817.474,A -85,B 0,C 180,E1 -4759.283,E2 -4759.283} C_VEL
LIN {X 0,Y 524.107,Z 826.34,A -85,B 0,C 180,E1 -4760.157,E2 -4760.157} C_VEL
LIN {X 0,Y 523.856,Z 834.483,A -85,B 0,C 180,E1 -4761.126,E2 -4761.126} C_VEL
LIN {X 0,Y 523.664,Z 842.471,A -85,B 0,C 180,E1 -4762.288,E2 -4762.288} C_VEL
LIN {X 0,Y 523.521,Z 848.736,A -85,B 0,C 180,E1 -4763.421,E2 -4763.421} C_VEL
LIN {X 0,Y 523.464,Z 853.951,A -85,B 0,C 180,E1 -4764.608,E2 -4764.608} C_VEL
LIN {X 0,Y 523.441,Z 857.897,A -85,B 0,C 180,E1 -4765.766,E2 -4765.766} C_VEL
LIN {X 0,Y 523.367,Z 860.811,A -85,B 0,C 180,E1 -4766.922,E2 -4766.922} C_VEL
LIN {X 0,Y 523.334,Z 862.197,A -85,B 0,C 180,E1 -4767.692,E2 -4767.692} C_VEL
LIN {X 0,Y 523.25,Z 863.786,A -85,B 0,C 180,E1 -4769.231,E2 -4769.231} C_VEL
LIN {X 0,Y 523.246,Z 864,A -85,B 0,C 180,E1 -4770.001,E2 -4770.001} C_VEL
LIN {X 0,Y 523.274,Z 863.181,A -85,B 0,C 180,E1 -4771.54,E2 -4771.54} C_VEL
LIN {X 0,Y 523.334,Z 862.192,A -85,B 0,C 180,E1 -4772.31,E2 -4772.31} C_VEL
LIN {X 0,Y 523.368,Z 860.805,A -85,B 0,C 180,E1 -4773.08,E2 -4773.08} C_VEL
LIN {X 0,Y 523.442,Z 857.893,A -85,B 0,C 180,E1 -4774.235,E2 -4774.235} C_VEL
LIN {X 0,Y 523.464,Z 853.948,A -85,B 0,C 180,E1 -4775.393,E2 -4775.393} C_VEL
LIN {X 0,Y 523.523,Z 848.726,A -85,B 0,C 180,E1 -4776.581,E2 -4776.581} C_VEL
LIN {X 0,Y 523.665,Z 842.462,A -85,B 0,C 180,E1 -4777.713,E2 -4777.713} C_VEL
LIN {X 0,Y 523.857,Z 834.473,A -85,B 0,C 180,E1 -4778.876,E2 -4778.876} C_VEL
LIN {X 0,Y 524.108,Z 826.328,A -85,B 0,C 180,E1 -4779.845,E2 -4779.845} C_VEL
LIN {X 0,Y 524.366,Z 816.392,A -85,B 0,C 180,E1 -4780.816,E2 -4780.816} C_VEL
LIN {X 0,Y 524.664,Z 805.181,A -85,B 0,C 180,E1 -4781.688,E2 -4781.688} C_VEL
LIN {X 0,Y 524.922,Z 794.118,A -85,B 0,C 180,E1 -4782.37,E2 -4782.37} C_VEL
LIN {X 0,Y 525.196,Z 781.781,A -85,B 0,C 180,E1 -4782.953,E2 -4782.953} C_VEL
LIN {X 0,Y 525.358,Z 768.777,A -85,B 0,C 180,E1 -4783.392,E2 -4783.392} C_VEL
LIN {X 0,Y 525.561,Z 754.996,A -85,B 0,C 180,E1 -4783.682,E2 -4783.682} C_VEL
LIN {X 0,Y 525.814,Z 658.698,A -85,B 0,C 180,E1 -4785.003,E2 -4785.003} C_VEL
LIN {X 0,Y 524.517,Z 649.943,A -85,B 0,C 180,E1 -4785.171,E2 -4785.171} C_VEL
LIN {X 0,Y 524.896,Z 627.276,A -85,B 0,C 180,E1 -4788.076,E2 -4788.076} C_VEL
LIN {X 0,Y 525.426,Z 604.808,A -85,B 0,C 180,E1 -4790.982,E2 -4790.982} C_VEL
LIN {X 0,Y 525.885,Z 581.556,A -85,B 0,C 180,E1 -4794.055,E2 -4794.055} C_VEL
LIN {X 0,Y 526.418,Z 560.732,A -85,B 0,C 180,E1 -4796.853,E2 -4796.853} C_VEL
LIN {X 0,Y 526.576,Z 547.156,A -85,B 0,C 180,E1 -4798.717,E2 -4798.717} C_VEL
LIN {X 0,Y 523.963,Z 535.221,A -85,B 0,C 180,E1 -4800.532,E2 -4800.532} C_VEL
LIN {X 0,Y 523.964,Z 535.215,A -85,B 0,C 180,E1 -4803.735,E2 -4803.735} C_VEL
LIN {X 0,Y 523.907,Z 535.223,A -85,B 0,C 180,E1 -4806.401,E2 -4806.401} C_VEL
LIN {X 0,Y 523.926,Z 535.227,A -85,B 0,C 180,E1 -4809.084,E2 -4809.084} C_VEL
LIN {X 0,Y 523.955,Z 535.214,A -85,B 0,C 180,E1 -4812.119,E2 -4812.119} C_VEL
LIN {X 0,Y 523.958,Z 535.22,A -85,B 0,C 180,E1 -4815.309,E2 -4815.309} C_VEL
LIN {X 0,Y 523.963,Z 535.212,A -85,B 0,C 180,E1 -4818.689,E2 -4818.689} C_VEL
LIN {X 0,Y 523.918,Z 535.218,A -85,B 0,C 180,E1 -4821.898,E2 -4821.898} C_VEL
LIN {X 0,Y 523.94,Z 535.218,A -85,B 0,C 180,E1 -4824.909,E2 -4824.909} C_VEL
LIN {X 0,Y 523.938,Z 535.216,A -85,B 0,C 180,E1 -4827.679,E2 -4827.679} C_VEL
LIN {X 0,Y 523.954,Z 535.213,A -85,B 0,C 180,E1 -4830.676,E2 -4830.676} C_VEL
LIN {X 0,Y 523.975,Z 535.212,A -85,B 0,C 180,E1 -4833.728,E2 -4833.728} C_VEL
LIN {X 0,Y 523.926,Z 535.214,A -85,B 0,C 180,E1 -4836.27,E2 -4836.27} C_VEL
LIN {X 0,Y 523.946,Z 535.216,A -85,B 0,C 180,E1 -4838.767,E2 -4838.767} C_VEL
LIN {X 0,Y 523.952,Z 535.218,A -85,B 0,C 180,E1 -4841.221,E2 -4841.221} C_VEL
LIN {X 0,Y 523.937,Z 535.222,A -85,B 0,C 180,E1 -4843.639,E2 -4843.639} C_VEL
LIN {X 0,Y 523.944,Z 535.217,A -85,B 0,C 180,E1 -4846.028,E2 -4846.028} C_VEL
LIN {X 0,Y 524.012,Z 535.202,A -85,B 0,C 180,E1 -4848.394,E2 -4848.394} C_VEL
LIN {X 0,Y 524.004,Z 535.212,A -85,B 0,C 180,E1 -4851.516,E2 -4851.516} C_VEL
LIN {X 0,Y 524.083,Z 535.197,A -85,B 0,C 180,E1 -4854.614,E2 -4854.614} C_VEL
LIN {X 0,Y 524.111,Z 535.196,A -85,B 0,C 180,E1 -4857.695,E2 -4857.695} C_VEL
LIN {X 0,Y 524.123,Z 535.193,A -85,B 0,C 180,E1 -4860.768,E2 -4860.768} C_VEL
LIN {X 0,Y 524.073,Z 535.199,A -85,B 0,C 180,E1 -4863.075,E2 -4863.075} C_VEL
LIN {X 0,Y 524.046,Z 535.204,A -85,B 0,C 180,E1 -4866.159,E2 -4866.159} C_VEL
LIN {X 0,Y 523.999,Z 535.21,A -85,B 0,C 180,E1 -4869.262,E2 -4869.262} C_VEL
LIN {X 0,Y 524.002,Z 535.211,A -85,B 0,C 180,E1 -4871.74,E2 -4871.74} C_VEL
LIN {X 0,Y 523.992,Z 535.209,A -85,B 0,C 180,E1 -4875.052,E2 -4875.052} C_VEL
LIN {X 0,Y 523.964,Z 535.216,A -85,B 0,C 180,E1 -4877.969,E2 -4877.969} C_VEL
LIN {X 0,Y 523.972,Z 535.213,A -85,B 0,C 180,E1 -4880.41,E2 -4880.41} C_VEL
LIN {X 0,Y 523.917,Z 535.218,A -85,B 0,C 180,E1 -4882.893,E2 -4882.893} C_VEL
LIN {X 0,Y 523.953,Z 535.211,A -85,B 0,C 180,E1 -4885.419,E2 -4885.419} C_VEL
LIN {X 0,Y 523.97,Z 535.22,A -85,B 0,C 180,E1 -4887.999,E2 -4887.999} C_VEL
LIN {X 0,Y 523.945,Z 535.212,A -85,B 0,C 180,E1 -4890.855,E2 -4890.855} C_VEL
LIN {X 0,Y 523.96,Z 535.218,A -85,B 0,C 180,E1 -4893.735,E2 -4893.735} C_VEL
LIN {X 0,Y 523.904,Z 535.227,A -85,B 0,C 180,E1 -4896.402,E2 -4896.402} C_VEL
LIN {X 0,Y 523.924,Z 535.217,A -85,B 0,C 180,E1 -4899.085,E2 -4899.085} C_VEL
LIN {X 0,Y 523.958,Z 535.223,A -85,B 0,C 180,E1 -4902.119,E2 -4902.119} C_VEL
LIN {X 0,Y 523.946,Z 535.215,A -85,B 0,C 180,E1 -4905.31,E2 -4905.31} C_VEL
LIN {X 0,Y 523.907,Z 535.215,A -85,B 0,C 180,E1 -4906.914,E2 -4906.914} C_VEL
LIN {X 0,Y 523.248,Z 535.297,A -85,B 0,C 180,E1 -4907.555,E2 -4907.555} C_VEL
LIN {X 0,Y 520.412,Z 535.663,A -85,B 0,C 180,E1 -4908.597,E2 -4908.597} C_VEL
LIN {X 0,Y 518.008,Z 535.97,A -85,B 0,C 180,E1 -4909.436,E2 -4909.436} C_VEL
LIN {X 0,Y 516.971,Z 536.096,A -85,B 0,C 180,E1 -4910.084,E2 -4910.084} C_VEL
LIN {X 0,Y 516.883,Z 536.103,A -85,B 0,C 180,E1 -4910.303,E2 -4910.303} C_VEL
LIN {X 0,Y 516.881,Z 536.096,A -85,B 0,C 180,E1 -4913.343,E2 -4913.343} C_VEL
LIN {X 0,Y 516.914,Z 536.098,A -85,B 0,C 180,E1 -4916.121,E2 -4916.121} C_VEL
LIN {X 0,Y 516.895,Z 536.101,A -85,B 0,C 180,E1 -4918.936,E2 -4918.936} C_VEL
LIN {X 0,Y 516.923,Z 536.094,A -85,B 0,C 180,E1 -4921.585,E2 -4921.585} C_VEL
LIN {X 0,Y 516.945,Z 536.202,A -85,B 0,C 180,E1 -4923.07,E2 -4923.07} C_VEL
LIN {X 0,Y 519.32,Z 547.734,A -85,B 0,C 180,E1 -4924.757,E2 -4924.757} C_VEL
LIN {X 0,Y 518.902,Z 565.545,A -85,B 0,C 180,E1 -4927.19,E2 -4927.19} C_VEL
LIN {X 0,Y 518.349,Z 589.145,A -85,B 0,C 180,E1 -4930.392,E2 -4930.392} C_VEL
LIN {X 0,Y 517.838,Z 611.858,A -85,B 0,C 180,E1 -4933.44,E2 -4933.44} C_VEL
LIN {X 0,Y 517.67,Z 621.338,A -85,B 0,C 180,E1 -4934.68,E2 -4934.68} C_VEL
LIN {X 0,Y 519.094,Z 631.643,A -85,B 0,C 180,E1 -4934.869,E2 -4934.869} C_VEL
LIN {X 0,Y 518.707,Z 730.232,A -85,B 0,C 180,E1 -4936.259,E2 -4936.259} C_VEL
LIN {X 0,Y 518.468,Z 742.855,A -85,B 0,C 180,E1 -4936.577,E2 -4936.577} C_VEL
LIN {X 0,Y 518.17,Z 755.705,A -85,B 0,C 180,E1 -4937.068,E2 -4937.068} C_VEL
LIN {X 0,Y 517.878,Z 768.47,A -85,B 0,C 180,E1 -4937.741,E2 -4937.741} C_VEL
LIN {X 0,Y 517.612,Z 780.123,A -85,B 0,C 180,E1 -4938.546,E2 -4938.546} C_VEL
LIN {X 0,Y 517.243,Z 790.339,A -85,B 0,C 180,E1 -4939.43,E2 -4939.43} C_VEL
LIN {X 0,Y 516.975,Z 799.586,A -85,B 0,C 180,E1 -4940.413,E2 -4940.413} C_VEL
LIN {X 0,Y 516.725,Z 808.503,A -85,B 0,C 180,E1 -4941.592,E2 -4941.592} C_VEL
LIN {X 0,Y 516.515,Z 815.671,A -85,B 0,C 180,E1 -4942.769,E2 -4942.769} C_VEL
LIN {X 0,Y 516.436,Z 820.542,A -85,B 0,C 180,E1 -4943.749,E2 -4943.749} C_VEL
LIN {X 0,Y 516.314,Z 825.255,A -85,B 0,C 180,E1 -4944.923,E2 -4944.923} C_VEL
LIN {X 0,Y 516.373,Z 828.859,A -85,B 0,C 180,E1 -4946.097,E2 -4946.097} C_VEL
LIN {X 0,Y 516.283,Z 830.718,A -85,B 0,C 180,E1 -4946.878,E2 -4946.878} C_VEL
LIN {X 0,Y 516.261,Z 832.143,A -85,B 0,C 180,E1 -4947.659,E2 -4947.659} C_VEL
LIN {X 0,Y 516.16,Z 833.759,A -85,B 0,C 180,E1 -4949.219,E2 -4949.219} C_VEL
LIN {X 0,Y 516.155,Z 833.998,A -85,B 0,C 180,E1 -4949.999,E2 -4949.999} C_VEL
LIN {X 0,Y 516.16,Z 833.814,A -85,B 0,C 180,E1 -4950.779,E2 -4950.779} C_VEL
LIN {X 0,Y 516.261,Z 832.272,A -85,B 0,C 180,E1 -4952.34,E2 -4952.34} C_VEL
LIN {X 0,Y 516.283,Z 830.918,A -85,B 0,C 180,E1 -4953.121,E2 -4953.121} C_VEL
LIN {X 0,Y 516.344,Z 828.064,A -85,B 0,C 180,E1 -4954.293,E2 -4954.293} C_VEL
LIN {X 0,Y 516.4,Z 824.186,A -85,B 0,C 180,E1 -4955.466,E2 -4955.466} C_VEL
LIN {X 0,Y 516.479,Z 818.386,A -85,B 0,C 180,E1 -4956.798,E2 -4956.798} C_VEL
LIN {X 0,Y 516.639,Z 811.646,A -85,B 0,C 180,E1 -4958.014,E2 -4958.014} C_VEL
LIN {X 0,Y 516.853,Z 803.504,A -85,B 0,C 180,E1 -4959.193,E2 -4959.193} C_VEL
LIN {X 0,Y 517.087,Z 795.118,A -85,B 0,C 180,E1 -4960.176,E2 -4960.176} C_VEL
LIN {X 0,Y 517.461,Z 784.84,A -85,B 0,C 180,E1 -4961.159,E2 -4961.159} C_VEL
LIN {X 0,Y 517.746,Z 774.253,A -85,B 0,C 180,E1 -4961.976,E2 -4961.976} C_VEL
LIN {X 0,Y 518.002,Z 763.467,A -85,B 0,C 180,E1 -4962.636,E2 -4962.636} C_VEL
LIN {X 0,Y 518.314,Z 750.865,A -85,B 0,C 180,E1 -4963.226,E2 -4963.226} C_VEL
LIN {X 0,Y 518.552,Z 738.438,A -85,B 0,C 180,E1 -4963.644,E2 -4963.644} C_VEL
LIN {X 0,Y 518.697,Z 725.614,A -85,B 0,C 180,E1 -4963.915,E2 -4963.915} C_VEL
LIN {X 0,Y 519.019,Z 631.443,A -85,B 0,C 180,E1 -4965.226,E2 -4965.226} C_VEL
LIN {X 0,Y 517.453,Z 621.537,A -85,B 0,C 180,E1 -4965.437,E2 -4965.437} C_VEL
LIN {X 0,Y 517.889,Z 602.176,A -85,B 0,C 180,E1 -4968.37,E2 -4968.37} C_VEL
LIN {X 0,Y 518.338,Z 582.971,A -85,B 0,C 180,E1 -4971.265,E2 -4971.265} C_VEL
LIN {X 0,Y 518.818,Z 563.789,A -85,B 0,C 180,E1 -4974.189,E2 -4974.189} C_VEL
LIN {X 0,Y 519.161,Z 547.558,A -85,B 0,C 180,E1 -4976.688,E2 -4976.688} C_VEL
LIN {X 0,Y 516.923,Z 536.098,A -85,B 0,C 180,E1 -4978.552,E2 -4978.552} C_VEL
LIN {X 0,Y 516.889,Z 536.102,A -85,B 0,C 180,E1 -4981.108,E2 -4981.108} C_VEL
LIN {X 0,Y 516.912,Z 536.095,A -85,B 0,C 180,E1 -4983.966,E2 -4983.966} C_VEL
LIN {X 0,Y 516.881,Z 536.097,A -85,B 0,C 180,E1 -4986.744,E2 -4986.744} C_VEL
LIN {X 0,Y 516.878,Z 536.099,A -85,B 0,C 180,E1 -4989.72,E2 -4989.72} C_VEL
LIN {X 0,Y 516.901,Z 536.094,A -85,B 0,C 180,E1 -4992.76,E2 -4992.76} C_VEL
LIN {X 0,Y 516.917,Z 536.092,A -85,B 0,C 180,E1 -4995.009,E2 -4995.009} C_VEL
LIN {X 0,Y 516.923,Z 536.091,A -85,B 0,C 180,E1 -4998.396,E2 -4998.396} C_VEL
LIN {X 0,Y 516.9,Z 536.101,A -85,B 0,C 180,E1 -5001.286,E2 -5001.286} C_VEL
LIN {X 0,Y 516.908,Z 536.099,A -85,B 0,C 180,E1 -5003.105,E2 -5003.105} C_VEL
LIN {X 0,Y 518.995,Z 542.487,A -85,B 0,C 180,E1 -5003.268,E2 -5003.268} C_VEL
LIN {X 0,Y 518.627,Z 616.208,A -85,B 0,C 180,E1 -5004.344,E2 -5004.344} C_VEL
LIN {X 0,Y 518.53,Z 628.771,A -85,B 0,C 180,E1 -5004.679,E2 -5004.679} C_VEL
LIN {X 0,Y 518.378,Z 641.334,A -85,B 0,C 180,E1 -5005.172,E2 -5005.172} C_VEL
LIN {X 0,Y 518.148,Z 653.583,A -85,B 0,C 180,E1 -5005.829,E2 -5005.829} C_VEL
LIN {X 0,Y 517.9,Z 664.011,A -85,B 0,C 180,E1 -5006.544,E2 -5006.544} C_VEL
LIN {X 0,Y 517.653,Z 674.21,A -85,B 0,C 180,E1 -5007.413,E2 -5007.413} C_VEL
LIN {X 0,Y 517.368,Z 684.18,A -85,B 0,C 180,E1 -5008.467,E2 -5008.467} C_VEL
LIN {X 0,Y 517.128,Z 692.664,A -85,B 0,C 180,E1 -5009.586,E2 -5009.586} C_VEL
LIN {X 0,Y 516.91,Z 699.506,A -85,B 0,C 180,E1 -5010.695,E2 -5010.695} C_VEL
LIN {X 0,Y 516.771,Z 705.482,A -85,B 0,C 180,E1 -5011.899,E2 -5011.899} C_VEL
LIN {X 0,Y 516.687,Z 710.888,A -85,B 0,C 180,E1 -5013.329,E2 -5013.329} C_VEL
LIN {X 0,Y 516.613,Z 713.401,A -85,B 0,C 180,E1 -5014.194,E2 -5014.194} C_VEL
LIN {X 0,Y 516.553,Z 715.364,A -85,B 0,C 180,E1 -5015.053,E2 -5015.053} C_VEL
LIN {X 0,Y 516.517,Z 716.805,A -85,B 0,C 180,E1 -5015.908,E2 -5015.908} C_VEL
LIN {X 0,Y 516.492,Z 717.791,A -85,B 0,C 180,E1 -5016.758,E2 -5016.758} C_VEL
LIN {X 0,Y 516.504,Z 718.288,A -85,B 0,C 180,E1 -5017.705,E2 -5017.705} C_VEL
LIN {X 0,Y 516.529,Z 717.909,A -85,B 0,C 180,E1 -5019.282,E2 -5019.282} C_VEL
LIN {X 0,Y 516.514,Z 717.035,A -85,B 0,C 180,E1 -5020.113,E2 -5020.113} C_VEL
LIN {X 0,Y 516.555,Z 715.728,A -85,B 0,C 180,E1 -5020.941,E2 -5020.941} C_VEL
LIN {X 0,Y 516.673,Z 712.832,A -85,B 0,C 180,E1 -5022.202,E2 -5022.202} C_VEL
LIN {X 0,Y 516.734,Z 708.995,A -85,B 0,C 180,E1 -5023.404,E2 -5023.404} C_VEL
LIN {X 0,Y 516.908,Z 703.977,A -85,B 0,C 180,E1 -5024.607,E2 -5024.607} C_VEL
LIN {X 0,Y 517.102,Z 697.406,A -85,B 0,C 180,E1 -5025.839,E2 -5025.839} C_VEL
LIN {X 0,Y 517.333,Z 689.305,A -85,B 0,C 180,E1 -5027.047,E2 -5027.047} C_VEL
LIN {X 0,Y 517.557,Z 680.789,A -85,B 0,C 180,E1 -5028.074,E2 -5028.074} C_VEL
LIN {X 0,Y 517.784,Z 670.819,A -85,B 0,C 180,E1 -5029.046,E2 -5029.046} C_VEL
LIN {X 0,Y 518.11,Z 659.216,A -85,B 0,C 180,E1 -5029.942,E2 -5029.942} C_VEL
LIN {X 0,Y 518.371,Z 647.693,A -85,B 0,C 180,E1 -5030.637,E2 -5030.637} C_VEL
LIN {X 0,Y 518.528,Z 635.771,A -85,B 0,C 180,E1 -5031.18,E2 -5031.18} C_VEL
LIN {X 0,Y 518.597,Z 622.622,A -85,B 0,C 180,E1 -5031.608,E2 -5031.608} C_VEL
LIN {X 0,Y 518.67,Z 609.626,A -85,B 0,C 180,E1 -5031.862,E2 -5031.862} C_VEL
LIN {X 0,Y 518.953,Z 542.348,A -85,B 0,C 180,E1 -5032.832,E2 -5032.832} C_VEL
LIN {X 0,Y 516.995,Z 536.089,A -85,B 0,C 180,E1 -5032.998,E2 -5032.998} C_VEL
LIN {X 0,Y 516.934,Z 536.092,A -85,B 0,C 180,E1 -5035.321,E2 -5035.321} C_VEL
LIN {X 0,Y 517.075,Z 536.073,A -85,B 0,C 180,E1 -5037.663,E2 -5037.663} C_VEL
LIN {X 0,Y 517.087,Z 536.079,A -85,B 0,C 180,E1 -5040.779,E2 -5040.779} C_VEL
LIN {X 0,Y 517.008,Z 536.083,A -85,B 0,C 180,E1 -5043.117,E2 -5043.117} C_VEL
LIN {X 0,Y 517.004,Z 536.083,A -85,B 0,C 180,E1 -5046.243,E2 -5046.243} C_VEL
LIN {X 0,Y 516.948,Z 536.087,A -85,B 0,C 180,E1 -5049.389,E2 -5049.389} C_VEL
LIN {X 0,Y 516.972,Z 536.085,A -85,B 0,C 180,E1 -5051.824,E2 -5051.824} C_VEL
LIN {X 0,Y 516.935,Z 536.09,A -85,B 0,C 180,E1 -5055.148,E2 -5055.148} C_VEL
LIN {X 0,Y 516.915,Z 536.093,A -85,B 0,C 180,E1 -5058.223,E2 -5058.223} C_VEL
LIN {X 0,Y 516.903,Z 536.101,A -85,B 0,C 180,E1 -5060.702,E2 -5060.702} C_VEL
LIN {X 0,Y 516.901,Z 536.094,A -85,B 0,C 180,E1 -5064.073,E2 -5064.073} C_VEL
LIN {X 0,Y 516.92,Z 536.097,A -85,B 0,C 180,E1 -5066.658,E2 -5066.658} C_VEL
LIN {X 0,Y 516.916,Z 536.092,A -85,B 0,C 180,E1 -5069.527,E2 -5069.527} C_VEL
LIN {X 0,Y 516.893,Z 536.1,A -85,B 0,C 180,E1 -5072.545,E2 -5072.545} C_VEL
LIN {X 0,Y 516.876,Z 536.099,A -85,B 0,C 180,E1 -5075.334,E2 -5075.334} C_VEL
LIN {X 0,Y 516.875,Z 536.095,A -85,B 0,C 180,E1 -5077.944,E2 -5077.944} C_VEL
LIN {X 0,Y 516.902,Z 536.099,A -85,B 0,C 180,E1 -5080.74,E2 -5080.74} C_VEL
LIN {X 0,Y 516.877,Z 536.097,A -85,B 0,C 180,E1 -5083.904,E2 -5083.904} C_VEL
LIN {X 0,Y 516.876,Z 536.098,A -85,B 0,C 180,E1 -5086.108,E2 -5086.108} C_VEL
LIN {X 0,Y 516.899,Z 536.098,A -85,B 0,C 180,E1 -5089.261,E2 -5089.261} C_VEL
LIN {X 0,Y 516.881,Z 536.097,A -85,B 0,C 180,E1 -5092.057,E2 -5092.057} C_VEL
LIN {X 0,Y 516.893,Z 536.101,A -85,B 0,C 180,E1 -5095.177,E2 -5095.177} C_VEL
LIN {X 0,Y 516.88,Z 536.098,A -85,B 0,C 180,E1 -5097.977,E2 -5097.977} C_VEL
LIN {X 0,Y 516.939,Z 536.141,A -85,B 0,C 180,E1 -5101.282,E2 -5101.282} C_VEL
LIN {X 0,Y 519.636,Z 548.741,A -85,B 0,C 180,E1 -5102.968,E2 -5102.968} C_VEL
LIN {X 0,Y 519.232,Z 568.874,A -85,B 0,C 180,E1 -5105.405,E2 -5105.405} C_VEL
LIN {X 0,Y 518.742,Z 591.806,A -85,B 0,C 180,E1 -5108.127,E2 -5108.127} C_VEL
LIN {X 0,Y 518.206,Z 618.434,A -85,B 0,C 180,E1 -5111.231,E2 -5111.231} C_VEL
LIN {X 0,Y 517.636,Z 647.918,A -85,B 0,C 180,E1 -5114.627,E2 -5114.627} C_VEL
LIN {X 0,Y 519.073,Z 661.058,A -85,B 0,C 180,E1 -5114.853,E2 -5114.853} C_VEL
LIN {X 0,Y 518.617,Z 757.64,A -85,B 0,C 180,E1 -5116.208,E2 -5116.208} C_VEL
LIN {X 0,Y 518.323,Z 771.36,A -85,B 0,C 180,E1 -5116.549,E2 -5116.549} C_VEL
LIN {X 0,Y 518.108,Z 784.963,A -85,B 0,C 180,E1 -5117.067,E2 -5117.067} C_VEL
LIN {X 0,Y 517.804,Z 797.423,A -85,B 0,C 180,E1 -5117.721,E2 -5117.721} C_VEL
LIN {X 0,Y 517.494,Z 809.572,A -85,B 0,C 180,E1 -5118.545,E2 -5118.545} C_VEL
LIN {X 0,Y 517.178,Z 819.98,A -85,B 0,C 180,E1 -5119.43,E2 -5119.43} C_VEL
LIN {X 0,Y 516.938,Z 829.383,A -85,B 0,C 180,E1 -5120.414,E2 -5120.414} C_VEL
LIN {X 0,Y 516.716,Z 838.526,A -85,B 0,C 180,E1 -5121.593,E2 -5121.593} C_VEL
LIN {X 0,Y 516.509,Z 845.812,A -85,B 0,C 180,E1 -5122.77,E2 -5122.77} C_VEL
LIN {X 0,Y 516.426,Z 850.679,A -85,B 0,C 180,E1 -5123.75,E2 -5123.75} C_VEL
LIN {X 0,Y 516.313,Z 855.374,A -85,B 0,C 180,E1 -5124.925,E2 -5124.925} C_VEL
LIN {X 0,Y 516.355,Z 858.962,A -85,B 0,C 180,E1 -5126.098,E2 -5126.098} C_VEL
LIN {X 0,Y 516.282,Z 860.811,A -85,B 0,C 180,E1 -5126.879,E2 -5126.879} C_VEL
LIN {X 0,Y 516.26,Z 862.196,A -85,B 0,C 180,E1 -5127.66,E2 -5127.66} C_VEL
LIN {X 0,Y 516.16,Z 863.786,A -85,B 0,C 180,E1 -5129.221,E2 -5129.221} C_VEL
LIN {X 0,Y 516.154,Z 864,A -85,B 0,C 180,E1 -5130.001,E2 -5130.001} C_VEL
LIN {X 0,Y 516.192,Z 863.181,A -85,B 0,C 180,E1 -5131.561,E2 -5131.561} C_VEL
LIN {X 0,Y 516.26,Z 862.192,A -85,B 0,C 180,E1 -5132.341,E2 -5132.341} C_VEL
LIN {X 0,Y 516.283,Z 860.805,A -85,B 0,C 180,E1 -5133.122,E2 -5133.122} C_VEL
LIN {X 0,Y 516.344,Z 857.892,A -85,B 0,C 180,E1 -5134.294,E2 -5134.294} C_VEL
LIN {X 0,Y 516.405,Z 853.948,A -85,B 0,C 180,E1 -5135.467,E2 -5135.467} C_VEL
LIN {X 0,Y 516.487,Z 848.013,A -85,B 0,C 180,E1 -5136.808,E2 -5136.808} C_VEL
LIN {X 0,Y 516.641,Z 841.12,A -85,B 0,C 180,E1 -5138.016,E2 -5138.016} C_VEL
LIN {X 0,Y 516.845,Z 832.68,A -85,B 0,C 180,E1 -5139.194,E2 -5139.194} C_VEL
LIN {X 0,Y 517.067,Z 824.014,A -85,B 0,C 180,E1 -5140.178,E2 -5140.178} C_VEL
LIN {X 0,Y 517.417,Z 813.35,A -85,B 0,C 180,E1 -5141.161,E2 -5141.161} C_VEL
LIN {X 0,Y 517.669,Z 801.623,A -85,B 0,C 180,E1 -5142.029,E2 -5142.029} C_VEL
LIN {X 0,Y 518,Z 789.265,A -85,B 0,C 180,E1 -5142.737,E2 -5142.737} C_VEL
LIN {X 0,Y 518.282,Z 776.716,A -85,B 0,C 180,E1 -5143.278,E2 -5143.278} C_VEL
LIN {X 0,Y 518.516,Z 763.765,A -85,B 0,C 180,E1 -5143.672,E2 -5143.672} C_VEL
LIN {X 0,Y 518.651,Z 748.396,A -85,B 0,C 180,E1 -5143.943,E2 -5143.943} C_VEL
LIN {X 0,Y 519.006,Z 659.922,A -85,B 0,C 180,E1 -5145.17,E2 -5145.17} C_VEL
LIN {X 0,Y 517.506,Z 649.013,A -85,B 0,C 180,E1 -5145.388,E2 -5145.388} C_VEL
LIN {X 0,Y 517.959,Z 624.734,A -85,B 0,C 180,E1 -5148.554,E2 -5148.554} C_VEL
LIN {X 0,Y 518.464,Z 604.178,A -85,B 0,C 180,E1 -5151.261,E2 -5151.261} C_VEL
LIN {X 0,Y 518.984,Z 580.795,A -85,B 0,C 180,E1 -5154.395,E2 -5154.395} C_VEL
LIN {X 0,Y 519.574,Z 558.963,A -85,B 0,C 180,E1 -5157.381,E2 -5157.381} C_VEL
LIN {X 0,Y 519.76,Z 549.106,A -85,B 0,C 180,E1 -5158.755,E2 -5158.755} C_VEL
LIN {X 0,Y 516.908,Z 536.1,A -85,B 0,C 180,E1 -5160.757,E2 -5160.757} C_VEL
LIN {X 0,Y 516.914,Z 536.093,A -85,B 0,C 180,E1 -5163.967,E2 -5163.967} C_VEL
LIN {X 0,Y 516.879,Z 536.102,A -85,B 0,C 180,E1 -5166.746,E2 -5166.746} C_VEL
LIN {X 0,Y 516.885,Z 536.096,A -85,B 0,C 180,E1 -5169.721,E2 -5169.721} C_VEL
LIN {X 0,Y 516.915,Z 536.092,A -85,B 0,C 180,E1 -5171.775,E2 -5171.775} C_VEL
LIN {X 0,Y 516.925,Z 536.094,A -85,B 0,C 180,E1 -5175.01,E2 -5175.01} C_VEL
LIN {X 0,Y 516.919,Z 536.087,A -85,B 0,C 180,E1 -5178.398,E2 -5178.398} C_VEL
LIN {X 0,Y 516.885,Z 536.102,A -85,B 0,C 180,E1 -5181.284,E2 -5181.284} C_VEL
LIN {X 0,Y 516.892,Z 536.091,A -85,B 0,C 180,E1 -5184.221,E2 -5184.221} C_VEL
LIN {X 0,Y 516.897,Z 536.099,A -85,B 0,C 180,E1 -5187.053,E2 -5187.053} C_VEL
LIN {X 0,Y 516.892,Z 536.094,A -85,B 0,C 180,E1 -5189.796,E2 -5189.796} C_VEL
LIN {X 0,Y 516.928,Z 536.089,A -85,B 0,C 180,E1 -5192.467,E2 -5192.467} C_VEL
LIN {X 0,Y 516.909,Z 536.093,A -85,B 0,C 180,E1 -5195.072,E2 -5195.072} C_VEL
LIN {X 0,Y 516.885,Z 536.094,A -85,B 0,C 180,E1 -5198.462,E2 -5198.462} C_VEL
LIN {X 0,Y 516.903,Z 536.093,A -85,B 0,C 180,E1 -5200.955,E2 -5200.955} C_VEL
LIN {X 0,Y 516.914,Z 536.092,A -85,B 0,C 180,E1 -5203.41,E2 -5203.41} C_VEL
LIN {X 0,Y 516.905,Z 536.096,A -85,B 0,C 180,E1 -5205.834,E2 -5205.834} C_VEL
LIN {X 0,Y 516.951,Z 536.084,A -85,B 0,C 180,E1 -5209.028,E2 -5209.028} C_VEL
LIN {X 0,Y 516.978,Z 536.084,A -85,B 0,C 180,E1 -5212.187,E2 -5212.187} C_VEL
LIN {X 0,Y 517.03,Z 536.076,A -85,B 0,C 180,E1 -5214.54,E2 -5214.54} C_VEL
LIN {X 0,Y 517.083,Z 536.07,A -85,B 0,C 180,E1 -5217.663,E2 -5217.663} C_VEL
LIN {X 0,Y 517.093,Z 536.068,A -85,B 0,C 180,E1 -5220.779,E2 -5220.779} C_VEL
LIN {X 0,Y 517.014,Z 536.078,A -85,B 0,C 180,E1 -5223.117,E2 -5223.117} C_VEL
LIN {X 0,Y 517.01,Z 536.079,A -85,B 0,C 180,E1 -5226.243,E2 -5226.243} C_VEL
LIN {X 0,Y 516.954,Z 536.089,A -85,B 0,C 180,E1 -5229.389,E2 -5229.389} C_VEL
LIN {X 0,Y 516.952,Z 536.088,A -85,B 0,C 180,E1 -5231.807,E2 -5231.807} C_VEL
LIN {X 0,Y 516.944,Z 536.087,A -85,B 0,C 180,E1 -5235.147,E2 -5235.147} C_VEL
LIN {X 0,Y 516.926,Z 536.088,A -85,B 0,C 180,E1 -5238.222,E2 -5238.222} C_VEL
LIN {X 0,Y 516.912,Z 536.09,A -85,B 0,C 180,E1 -5240.702,E2 -5240.702} C_VEL
LIN {X 0,Y 516.912,Z 536.095,A -85,B 0,C 180,E1 -5244.072,E2 -5244.072} C_VEL
LIN {X 0,Y 516.926,Z 536.09,A -85,B 0,C 180,E1 -5246.658,E2 -5246.658} C_VEL
LIN {X 0,Y 516.911,Z 536.093,A -85,B 0,C 180,E1 -5249.524,E2 -5249.524} C_VEL
LIN {X 0,Y 516.896,Z 536.097,A -85,B 0,C 180,E1 -5252.543,E2 -5252.543} C_VEL
LIN {X 0,Y 516.867,Z 536.095,A -85,B 0,C 180,E1 -5255.33,E2 -5255.33} C_VEL
LIN {X 0,Y 516.883,Z 536.102,A -85,B 0,C 180,E1 -5257.943,E2 -5257.943} C_VEL
LIN {X 0,Y 516.887,Z 536.097,A -85,B 0,C 180,E1 -5260.742,E2 -5260.742} C_VEL
LIN {X 0,Y 516.886,Z 536.094,A -85,B 0,C 180,E1 -5262.831,E2 -5262.831} C_VEL
LIN {X 0,Y 516.897,Z 536.094,A -85,B 0,C 180,E1 -5265.007,E2 -5265.007} C_VEL
LIN {X 0,Y 516.915,Z 536.095,A -85,B 0,C 180,E1 -5268.399,E2 -5268.399} C_VEL
LIN {X 0,Y 516.883,Z 536.103,A -85,B 0,C 180,E1 -5270.303,E2 -5270.303} C_VEL
LIN {X 0,Y 516.212,Z 536.18,A -85,B 0,C 180,E1 -5270.953,E2 -5270.953} C_VEL
LIN {X 0,Y 513.364,Z 536.535,A -85,B 0,C 180,E1 -5272.009,E2 -5272.009} C_VEL
LIN {X 0,Y 510.956,Z 536.836,A -85,B 0,C 180,E1 -5272.859,E2 -5272.859} C_VEL
LIN {X 0,Y 509.915,Z 536.965,A -85,B 0,C 180,E1 -5273.516,E2 -5273.516} C_VEL
LIN {X 0,Y 509.826,Z 536.976,A -85,B 0,C 180,E1 -5273.738,E2 -5273.738} C_VEL
LIN {X 0,Y 509.865,Z 536.978,A -85,B 0,C 180,E1 -5276.539,E2 -5276.539} C_VEL
LIN {X 0,Y 509.849,Z 536.976,A -85,B 0,C 180,E1 -5279.334,E2 -5279.334} C_VEL
LIN {X 0,Y 509.902,Z 536.974,A -85,B 0,C 180,E1 -5282.501,E2 -5282.501} C_VEL
LIN {X 0,Y 509.91,Z 537.114,A -85,B 0,C 180,E1 -5282.862,E2 -5282.862} C_VEL
LIN {X 0,Y 512.408,Z 549.029,A -85,B 0,C 180,E1 -5284.621,E2 -5284.621} C_VEL
LIN {X 0,Y 512.144,Z 562.957,A -85,B 0,C 180,E1 -5286.549,E2 -5286.549} C_VEL
LIN {X 0,Y 511.465,Z 585.957,A -85,B 0,C 180,E1 -5289.708,E2 -5289.708} C_VEL
LIN {X 0,Y 510.978,Z 607.253,A -85,B 0,C 180,E1 -5292.593,E2 -5292.593} C_VEL
LIN {X 0,Y 510.744,Z 621.55,A -85,B 0,C 180,E1 -5294.469,E2 -5294.469} C_VEL
LIN {X 0,Y 512.244,Z 631.926,A -85,B 0,C 180,E1 -5294.664,E2 -5294.664} C_VEL
LIN {X 0,Y 511.819,Z 730.348,A -85,B 0,C 180,E1 -5296.07,E2 -5296.07} C_VEL
LIN {X 0,Y 511.568,Z 743.004,A -85,B 0,C 180,E1 -5296.392,E2 -5296.392} C_VEL
LIN {X 0,Y 511.272,Z 755.873,A -85,B 0,C 180,E1 -5296.89,E2 -5296.89} C_VEL
LIN {X 0,Y 510.963,Z 768.644,A -85,B 0,C 180,E1 -5297.572,E2 -5297.572} C_VEL
LIN {X 0,Y 510.679,Z 779.052,A -85,B 0,C 180,E1 -5298.288,E2 -5298.288} C_VEL
LIN {X 0,Y 510.301,Z 789.497,A -85,B 0,C 180,E1 -5299.184,E2 -5299.184} C_VEL
LIN {X 0,Y 509.97,Z 799.776,A -85,B 0,C 180,E1 -5300.28,E2 -5300.28} C_VEL
LIN {X 0,Y 509.698,Z 808.695,A -85,B 0,C 180,E1 -5301.475,E2 -5301.475} C_VEL
LIN {X 0,Y 509.48,Z 815.864,A -85,B 0,C 180,E1 -5302.669,E2 -5302.669} C_VEL
LIN {X 0,Y 509.368,Z 820.736,A -85,B 0,C 180,E1 -5303.662,E2 -5303.662} C_VEL
LIN {X 0,Y 509.248,Z 825.449,A -85,B 0,C 180,E1 -5304.853,E2 -5304.853} C_VEL
LIN {X 0,Y 509.301,Z 829.052,A -85,B 0,C 180,E1 -5306.043,E2 -5306.043} C_VEL
LIN {X 0,Y 509.202,Z 830.912,A -85,B 0,C 180,E1 -5306.835,E2 -5306.835} C_VEL
LIN {X 0,Y 509.19,Z 832.336,A -85,B 0,C 180,E1 -5307.626,E2 -5307.626} C_VEL
LIN {X 0,Y 509.074,Z 833.952,A -85,B 0,C 180,E1 -5309.208,E2 -5309.208} C_VEL
LIN {X 0,Y 509.066,Z 834.191,A -85,B 0,C 180,E1 -5309.999,E2 -5309.999} C_VEL
LIN {X 0,Y 509.073,Z 834.007,A -85,B 0,C 180,E1 -5310.79,E2 -5310.79} C_VEL
LIN {X 0,Y 509.19,Z 832.464,A -85,B 0,C 180,E1 -5312.372,E2 -5312.372} C_VEL
LIN {X 0,Y 509.202,Z 831.109,A -85,B 0,C 180,E1 -5313.164,E2 -5313.164} C_VEL
LIN {X 0,Y 509.269,Z 828.254,A -85,B 0,C 180,E1 -5314.352,E2 -5314.352} C_VEL
LIN {X 0,Y 509.337,Z 824.375,A -85,B 0,C 180,E1 -5315.542,E2 -5315.542} C_VEL
LIN {X 0,Y 509.384,Z 819.358,A -85,B 0,C 180,E1 -5316.734,E2 -5316.734} C_VEL
LIN {X 0,Y 509.589,Z 813.025,A -85,B 0,C 180,E1 -5317.926,E2 -5317.926} C_VEL
LIN {X 0,Y 509.769,Z 805.154,A -85,B 0,C 180,E1 -5319.122,E2 -5319.122} C_VEL
LIN {X 0,Y 510.028,Z 797.112,A -85,B 0,C 180,E1 -5320.118,E2 -5320.118} C_VEL
LIN {X 0,Y 510.415,Z 787.264,A -85,B 0,C 180,E1 -5321.114,E2 -5321.114} C_VEL
LIN {X 0,Y 510.739,Z 775.834,A -85,B 0,C 180,E1 -5322.039,E2 -5322.039} C_VEL
LIN {X 0,Y 511.045,Z 765.415,A -85,B 0,C 180,E1 -5322.71,E2 -5322.71} C_VEL
LIN {X 0,Y 511.354,Z 753.403,A -85,B 0,C 180,E1 -5323.309,E2 -5323.309} C_VEL
LIN {X 0,Y 511.616,Z 740.219,A -85,B 0,C 180,E1 -5323.782,E2 -5323.782} C_VEL
LIN {X 0,Y 511.786,Z 727.18,A -85,B 0,C 180,E1 -5324.082,E2 -5324.082} C_VEL
LIN {X 0,Y 512.291,Z 633.178,A -85,B 0,C 180,E1 -5325.407,E2 -5325.407} C_VEL
LIN {X 0,Y 510.48,Z 621.716,A -85,B 0,C 180,E1 -5325.65,E2 -5325.65} C_VEL
LIN {X 0,Y 510.993,Z 600.525,A -85,B 0,C 180,E1 -5328.856,E2 -5328.856} C_VEL
LIN {X 0,Y 511.423,Z 582.702,A -85,B 0,C 180,E1 -5331.567,E2 -5331.567} C_VEL
LIN {X 0,Y 511.917,Z 563.629,A -85,B 0,C 180,E1 -5334.512,E2 -5334.512} C_VEL
LIN {X 0,Y 512.292,Z 549.241,A -85,B 0,C 180,E1 -5336.752,E2 -5336.752} C_VEL
LIN {X 0,Y 509.886,Z 536.975,A -85,B 0,C 180,E1 -5338.754,E2 -5338.754} C_VEL
LIN {X 0,Y 509.824,Z 536.98,A -85,B 0,C 180,E1 -5341.589,E2 -5341.589} C_VEL
LIN {X 0,Y 509.852,Z 536.974,A -85,B 0,C 180,E1 -5344.412,E2 -5344.412} C_VEL
LIN {X 0,Y 509.819,Z 536.986,A -85,B 0,C 180,E1 -5347.339,E2 -5347.339} C_VEL
LIN {X 0,Y 509.834,Z 536.973,A -85,B 0,C 180,E1 -5350.381,E2 -5350.381} C_VEL
LIN {X 0,Y 509.835,Z 536.976,A -85,B 0,C 180,E1 -5353.063,E2 -5353.063} C_VEL
LIN {X 0,Y 509.826,Z 536.978,A -85,B 0,C 180,E1 -5355.791,E2 -5355.791} C_VEL
LIN {X 0,Y 509.865,Z 536.971,A -85,B 0,C 180,E1 -5358.575,E2 -5358.575} C_VEL
LIN {X 0,Y 509.85,Z 536.977,A -85,B 0,C 180,E1 -5361.785,E2 -5361.785} C_VEL
LIN {X 0,Y 509.873,Z 537.009,A -85,B 0,C 180,E1 -5362.909,E2 -5362.909} C_VEL
LIN {X 0,Y 512.213,Z 544.169,A -85,B 0,C 180,E1 -5363.088,E2 -5363.088} C_VEL
LIN {X 0,Y 511.737,Z 617.279,A -85,B 0,C 180,E1 -5364.172,E2 -5364.172} C_VEL
LIN {X 0,Y 511.668,Z 629.724,A -85,B 0,C 180,E1 -5364.511,E2 -5364.511} C_VEL
LIN {X 0,Y 511.49,Z 642.98,A -85,B 0,C 180,E1 -5365.042,E2 -5365.042} C_VEL
LIN {X 0,Y 511.226,Z 654.794,A -85,B 0,C 180,E1 -5365.692,E2 -5365.692} C_VEL
LIN {X 0,Y 510.959,Z 666.265,A -85,B 0,C 180,E1 -5366.502,E2 -5366.502} C_VEL
LIN {X 0,Y 510.686,Z 676.251,A -85,B 0,C 180,E1 -5367.383,E2 -5367.383} C_VEL
LIN {X 0,Y 510.388,Z 685.947,A -85,B 0,C 180,E1 -5368.449,E2 -5368.449} C_VEL
LIN {X 0,Y 510.151,Z 694.312,A -85,B 0,C 180,E1 -5369.584,E2 -5369.584} C_VEL
LIN {X 0,Y 509.917,Z 701.04,A -85,B 0,C 180,E1 -5370.706,E2 -5370.706} C_VEL
LIN {X 0,Y 509.747,Z 707.389,A -85,B 0,C 180,E1 -5372.046,E2 -5372.046} C_VEL
LIN {X 0,Y 509.675,Z 712.109,A -85,B 0,C 180,E1 -5373.35,E2 -5373.35} C_VEL
LIN {X 0,Y 509.55,Z 715.658,A -85,B 0,C 180,E1 -5374.686,E2 -5374.686} C_VEL
LIN {X 0,Y 509.506,Z 717.328,A -85,B 0,C 180,E1 -5375.555,E2 -5375.555} C_VEL
LIN {X 0,Y 509.481,Z 718.454,A -85,B 0,C 180,E1 -5376.419,E2 -5376.419} C_VEL
LIN {X 0,Y 509.469,Z 719.258,A -85,B 0,C 180,E1 -5377.551,E2 -5377.551} C_VEL
LIN {X 0,Y 509.483,Z 719.104,A -85,B 0,C 180,E1 -5378.982,E2 -5378.982} C_VEL
LIN {X 0,Y 509.527,Z 718.428,A -85,B 0,C 180,E1 -5379.828,E2 -5379.828} C_VEL
LIN {X 0,Y 509.545,Z 717.291,A -85,B 0,C 180,E1 -5380.669,E2 -5380.669} C_VEL
LIN {X 0,Y 509.646,Z 714.319,A -85,B 0,C 180,E1 -5382.079,E2 -5382.079} C_VEL
LIN {X 0,Y 509.781,Z 709.632,A -85,B 0,C 180,E1 -5383.583,E2 -5383.583} C_VEL
LIN {X 0,Y 509.996,Z 703.373,A -85,B 0,C 180,E1 -5385.026,E2 -5385.026} C_VEL
LIN {X 0,Y 510.197,Z 696.538,A -85,B 0,C 180,E1 -5386.254,E2 -5386.254} C_VEL
LIN {X 0,Y 510.419,Z 689.529,A -85,B 0,C 180,E1 -5387.273,E2 -5387.273} C_VEL
LIN {X 0,Y 510.659,Z 681.046,A -85,B 0,C 180,E1 -5388.288,E2 -5388.288} C_VEL
LIN {X 0,Y 510.953,Z 670.53,A -85,B 0,C 180,E1 -5389.299,E2 -5389.299} C_VEL
LIN {X 0,Y 511.225,Z 660.092,A -85,B 0,C 180,E1 -5390.105,E2 -5390.105} C_VEL
LIN {X 0,Y 511.501,Z 648.494,A -85,B 0,C 180,E1 -5390.809,E2 -5390.809} C_VEL
LIN {X 0,Y 511.65,Z 637.786,A -85,B 0,C 180,E1 -5391.31,E2 -5391.31} C_VEL
LIN {X 0,Y 511.728,Z 624.724,A -85,B 0,C 180,E1 -5391.751,E2 -5391.751} C_VEL
LIN {X 0,Y 511.782,Z 612.099,A -85,B 0,C 180,E1 -5392.018,E2 -5392.018} C_VEL
LIN {X 0,Y 512.176,Z 543.919,A -85,B 0,C 180,E1 -5393.019,E2 -5393.019} C_VEL
LIN {X 0,Y 509.934,Z 536.967,A -85,B 0,C 180,E1 -5393.201,E2 -5393.201} C_VEL
LIN {X 0,Y 509.904,Z 536.968,A -85,B 0,C 180,E1 -5395.256,E2 -5395.256} C_VEL
LIN {X 0,Y 510.047,Z 536.948,A -85,B 0,C 180,E1 -5397.631,E2 -5397.631} C_VEL
LIN {X 0,Y 510.056,Z 536.955,A -85,B 0,C 180,E1 -5400.789,E2 -5400.789} C_VEL
LIN {X 0,Y 509.951,Z 536.962,A -85,B 0,C 180,E1 -5403.16,E2 -5403.16} C_VEL
LIN {X 0,Y 509.972,Z 536.96,A -85,B 0,C 180,E1 -5406.33,E2 -5406.33} C_VEL
LIN {X 0,Y 509.908,Z 536.973,A -85,B 0,C 180,E1 -5408.72,E2 -5408.72} C_VEL
LIN {X 0,Y 509.94,Z 536.961,A -85,B 0,C 180,E1 -5411.931,E2 -5411.931} C_VEL
LIN {X 0,Y 509.882,Z 536.967,A -85,B 0,C 180,E1 -5415.242,E2 -5415.242} C_VEL
LIN {X 0,Y 509.878,Z 536.969,A -85,B 0,C 180,E1 -5418.002,E2 -5418.002} C_VEL
LIN {X 0,Y 509.84,Z 536.978,A -85,B 0,C 180,E1 -5421.002,E2 -5421.002} C_VEL
LIN {X 0,Y 509.827,Z 536.975,A -85,B 0,C 180,E1 -5423.564,E2 -5423.564} C_VEL
LIN {X 0,Y 509.904,Z 536.968,A -85,B 0,C 180,E1 -5426.38,E2 -5426.38} C_VEL
LIN {X 0,Y 509.877,Z 536.975,A -85,B 0,C 180,E1 -5428.844,E2 -5428.844} C_VEL
LIN {X 0,Y 509.817,Z 536.976,A -85,B 0,C 180,E1 -5431.59,E2 -5431.59} C_VEL
LIN {X 0,Y 509.847,Z 536.975,A -85,B 0,C 180,E1 -5434.414,E2 -5434.414} C_VEL
LIN {X 0,Y 509.813,Z 536.977,A -85,B 0,C 180,E1 -5437.341,E2 -5437.341} C_VEL
LIN {X 0,Y 509.856,Z 536.973,A -85,B 0,C 180,E1 -5440.381,E2 -5440.381} C_VEL
LIN {X 0,Y 509.835,Z 536.981,A -85,B 0,C 180,E1 -5443.065,E2 -5443.065} C_VEL
LIN {X 0,Y 509.824,Z 536.976,A -85,B 0,C 180,E1 -5445.793,E2 -5445.793} C_VEL
LIN {X 0,Y 509.861,Z 536.976,A -85,B 0,C 180,E1 -5448.577,E2 -5448.577} C_VEL
LIN {X 0,Y 509.854,Z 536.972,A -85,B 0,C 180,E1 -5451.786,E2 -5451.786} C_VEL
LIN {X 0,Y 509.844,Z 536.981,A -85,B 0,C 180,E1 -5454.624,E2 -5454.624} C_VEL
LIN {X 0,Y 509.864,Z 536.974,A -85,B 0,C 180,E1 -5457.482,E2 -5457.482} C_VEL
LIN {X 0,Y 509.889,Z 536.975,A -85,B 0,C 180,E1 -5460.932,E2 -5460.932} C_VEL
LIN {X 0,Y 509.93,Z 537.238,A -85,B 0,C 180,E1 -5461.104,E2 -5461.104} C_VEL
LIN {X 0,Y 512.744,Z 550.266,A -85,B 0,C 180,E1 -5462.887,E2 -5462.887} C_VEL
LIN {X 0,Y 512.288,Z 569.6,A -85,B 0,C 180,E1 -5465.266,E2 -5465.266} C_VEL
LIN {X 0,Y 511.733,Z 592.477,A -85,B 0,C 180,E1 -5468.023,E2 -5468.023} C_VEL
LIN {X 0,Y 511.112,Z 620.653,A -85,B 0,C 180,E1 -5471.356,E2 -5471.356} C_VEL
LIN {X 0,Y 510.581,Z 646.963,A -85,B 0,C 180,E1 -5474.412,E2 -5474.412} C_VEL
LIN {X 0,Y 512.182,Z 662.093,A -85,B 0,C 180,E1 -5474.679,E2 -5474.679} C_VEL
LIN {X 0,Y 511.687,Z 757.19,A -85,B 0,C 180,E1 -5476.042,E2 -5476.042} C_VEL
LIN {X 0,Y 511.362,Z 770.625,A -85,B 0,C 180,E1 -5476.388,E2 -5476.388} C_VEL
LIN {X 0,Y 511.121,Z 783.558,A -85,B 0,C 180,E1 -5476.888,E2 -5476.888} C_VEL
LIN {X 0,Y 510.805,Z 795.68,A -85,B 0,C 180,E1 -5477.523,E2 -5477.523} C_VEL
LIN {X 0,Y 510.517,Z 807.018,A -85,B 0,C 180,E1 -5478.285,E2 -5478.285} C_VEL
LIN {X 0,Y 510.194,Z 817.721,A -85,B 0,C 180,E1 -5479.183,E2 -5479.183} C_VEL
LIN {X 0,Y 509.947,Z 826.472,A -85,B 0,C 180,E1 -5480.081,E2 -5480.081} C_VEL
LIN {X 0,Y 509.712,Z 834.551,A -85,B 0,C 180,E1 -5481.077,E2 -5481.077} C_VEL
LIN {X 0,Y 509.512,Z 842.51,A -85,B 0,C 180,E1 -5482.272,E2 -5482.272} C_VEL
LIN {X 0,Y 509.339,Z 849.806,A -85,B 0,C 180,E1 -5483.663,E2 -5483.663} C_VEL
LIN {X 0,Y 509.248,Z 854.662,A -85,B 0,C 180,E1 -5484.854,E2 -5484.854} C_VEL
LIN {X 0,Y 509.286,Z 858.393,A -85,B 0,C 180,E1 -5486.044,E2 -5486.044} C_VEL
LIN {X 0,Y 509.2,Z 860.289,A -85,B 0,C 180,E1 -5486.836,E2 -5486.836} C_VEL
LIN {X 0,Y 509.189,Z 861.735,A -85,B 0,C 180,E1 -5487.628,E2 -5487.628} C_VEL
LIN {X 0,Y 509.073,Z 863.37,A -85,B 0,C 180,E1 -5489.21,E2 -5489.21} C_VEL
LIN {X 0,Y 509.066,Z 863.591,A -85,B 0,C 180,E1 -5490.001,E2 -5490.001} C_VEL
LIN {X 0,Y 509.073,Z 863.371,A -85,B 0,C 180,E1 -5490.792,E2 -5490.792} C_VEL
LIN {X 0,Y 509.189,Z 861.74,A -85,B 0,C 180,E1 -5492.374,E2 -5492.374} C_VEL
LIN {X 0,Y 509.201,Z 860.303,A -85,B 0,C 180,E1 -5493.165,E2 -5493.165} C_VEL
LIN {X 0,Y 509.252,Z 857.299,A -85,B 0,C 180,E1 -5494.354,E2 -5494.354} C_VEL
LIN {X 0,Y 509.344,Z 853.233,A -85,B 0,C 180,E1 -5495.543,E2 -5495.543} C_VEL
LIN {X 0,Y 509.417,Z 847.328,A -85,B 0,C 180,E1 -5496.865,E2 -5496.865} C_VEL
LIN {X 0,Y 509.573,Z 840.136,A -85,B 0,C 180,E1 -5498.128,E2 -5498.128} C_VEL
LIN {X 0,Y 509.783,Z 831.636,A -85,B 0,C 180,E1 -5499.323,E2 -5499.323} C_VEL
LIN {X 0,Y 510.035,Z 822.956,A -85,B 0,C 180,E1 -5500.32,E2 -5500.32} C_VEL
LIN {X 0,Y 510.361,Z 812.293,A -85,B 0,C 180,E1 -5501.317,E2 -5501.317} C_VEL
LIN {X 0,Y 510.62,Z 801.943,A -85,B 0,C 180,E1 -5502.1,E2 -5502.1} C_VEL
LIN {X 0,Y 510.968,Z 790.094,A -85,B 0,C 180,E1 -5502.815,E2 -5502.815} C_VEL
LIN {X 0,Y 511.281,Z 778.148,A -85,B 0,C 180,E1 -5503.362,E2 -5503.362} C_VEL
LIN {X 0,Y 511.513,Z 765.251,A -85,B 0,C 180,E1 -5503.786,E2 -5503.786} C_VEL
LIN {X 0,Y 511.7,Z 751.972,A -85,B 0,C 180,E1 -5504.06,E2 -5504.06} C_VEL
LIN {X 0,Y 512.156,Z 661.024,A -85,B 0,C 180,E1 -5505.345,E2 -5505.345} C_VEL
LIN {X 0,Y 510.479,Z 648.123,A -85,B 0,C 180,E1 -5505.607,E2 -5505.607} C_VEL
LIN {X 0,Y 510.983,Z 623.583,A -85,B 0,C 180,E1 -5508.858,E2 -5508.858} C_VEL
LIN {X 0,Y 511.468,Z 603.376,A -85,B 0,C 180,E1 -5511.566,E2 -5511.566} C_VEL
LIN {X 0,Y 512.034,Z 581.653,A -85,B 0,C 180,E1 -5514.524,E2 -5514.524} C_VEL
LIN {X 0,Y 512.699,Z 559.813,A -85,B 0,C 180,E1 -5517.558,E2 -5517.558} C_VEL
LIN {X 0,Y 512.861,Z 550.45,A -85,B 0,C 180,E1 -5518.885,E2 -5518.885} C_VEL
LIN {X 0,Y 509.859,Z 536.978,A -85,B 0,C 180,E1 -5521.016,E2 -5521.016} C_VEL
LIN {X 0,Y 509.864,Z 536.974,A -85,B 0,C 180,E1 -5523.461,E2 -5523.461} C_VEL
LIN {X 0,Y 509.828,Z 536.976,A -85,B 0,C 180,E1 -5526.353,E2 -5526.353} C_VEL
LIN {X 0,Y 509.85,Z 536.976,A -85,B 0,C 180,E1 -5529.352,E2 -5529.352} C_VEL
LIN {X 0,Y 509.836,Z 536.975,A -85,B 0,C 180,E1 -5532.49,E2 -5532.49} C_VEL
LIN {X 0,Y 509.859,Z 536.976,A -85,B 0,C 180,E1 -5535.332,E2 -5535.332} C_VEL
LIN {X 0,Y 509.86,Z 536.968,A -85,B 0,C 180,E1 -5538.575,E2 -5538.575} C_VEL
LIN {X 0,Y 509.853,Z 536.971,A -85,B 0,C 180,E1 -5541.786,E2 -5541.786} C_VEL
LIN {X 0,Y 509.847,Z 536.97,A -85,B 0,C 180,E1 -5544.623,E2 -5544.623} C_VEL
LIN {X 0,Y 509.864,Z 536.972,A -85,B 0,C 180,E1 -5547.481,E2 -5547.481} C_VEL
LIN {X 0,Y 509.859,Z 536.968,A -85,B 0,C 180,E1 -5550.274,E2 -5550.274} C_VEL
LIN {X 0,Y 509.885,Z 536.97,A -85,B 0,C 180,E1 -5552.944,E2 -5552.944} C_VEL
LIN {X 0,Y 509.864,Z 536.971,A -85,B 0,C 180,E1 -5555.574,E2 -5555.574} C_VEL
LIN {X 0,Y 509.85,Z 536.974,A -85,B 0,C 180,E1 -5558.998,E2 -5558.998} C_VEL
LIN {X 0,Y 509.888,Z 536.961,A -85,B 0,C 180,E1 -5561.999,E2 -5561.999} C_VEL
LIN {X 0,Y 509.91,Z 536.963,A -85,B 0,C 180,E1 -5564.819,E2 -5564.819} C_VEL
LIN {X 0,Y 509.9,Z 536.961,A -85,B 0,C 180,E1 -5568.124,E2 -5568.124} C_VEL
LIN {X 0,Y 509.916,Z 536.962,A -85,B 0,C 180,E1 -5571.28,E2 -5571.28} C_VEL
LIN {X 0,Y 509.978,Z 536.963,A -85,B 0,C 180,E1 -5573.67,E2 -5573.67} C_VEL
LIN {X 0,Y 510.054,Z 536.945,A -85,B 0,C 180,E1 -5577.631,E2 -5577.631} C_VEL
LIN {X 0,Y 510.063,Z 536.944,A -85,B 0,C 180,E1 -5580.79,E2 -5580.79} C_VEL
LIN {X 0,Y 509.956,Z 536.958,A -85,B 0,C 180,E1 -5583.16,E2 -5583.16} C_VEL
LIN {X 0,Y 509.978,Z 536.954,A -85,B 0,C 180,E1 -5586.33,E2 -5586.33} C_VEL
LIN {X 0,Y 509.916,Z 536.963,A -85,B 0,C 180,E1 -5588.72,E2 -5588.72} C_VEL
LIN {X 0,Y 509.904,Z 536.964,A -85,B 0,C 180,E1 -5591.932,E2 -5591.932} C_VEL
LIN {X 0,Y 509.894,Z 536.966,A -85,B 0,C 180,E1 -5595.242,E2 -5595.242} C_VEL
LIN {X 0,Y 509.889,Z 536.968,A -85,B 0,C 180,E1 -5598.001,E2 -5598.001} C_VEL
LIN {X 0,Y 509.85,Z 536.969,A -85,B 0,C 180,E1 -5601.002,E2 -5601.002} C_VEL
LIN {X 0,Y 509.87,Z 536.967,A -85,B 0,C 180,E1 -5604.426,E2 -5604.426} C_VEL
LIN {X 0,Y 509.885,Z 536.966,A -85,B 0,C 180,E1 -5607.056,E2 -5607.056} C_VEL
LIN {X 0,Y 509.858,Z 536.974,A -85,B 0,C 180,E1 -5609.751,E2 -5609.751} C_VEL
LIN {X 0,Y 509.873,Z 536.97,A -85,B 0,C 180,E1 -5612.774,E2 -5612.774} C_VEL
LIN {X 0,Y 509.826,Z 536.974,A -85,B 0,C 180,E1 -5615.579,E2 -5615.579} C_VEL
LIN {X 0,Y 509.852,Z 536.977,A -85,B 0,C 180,E1 -5618.338,E2 -5618.338} C_VEL
LIN {X 0,Y 509.86,Z 536.971,A -85,B 0,C 180,E1 -5621.425,E2 -5621.425} C_VEL
LIN {X 0,Y 509.841,Z 536.976,A -85,B 0,C 180,E1 -5624.67,E2 -5624.67} C_VEL
LIN {X 0,Y 509.855,Z 536.969,A -85,B 0,C 180,E1 -5628.104,E2 -5628.104} C_VEL
LIN {X 0,Y 509.848,Z 536.974,A -85,B 0,C 180,E1 -5630.648,E2 -5630.648} C_VEL
LIN {X 0,Y 509.826,Z 536.976,A -85,B 0,C 180,E1 -5633.738,E2 -5633.738} C_VEL
LIN {X 0,Y 509.16,Z 537.065,A -85,B 0,C 180,E1 -5634.398,E2 -5634.398} C_VEL
LIN {X 0,Y 506.346,Z 537.413,A -85,B 0,C 180,E1 -5635.47,E2 -5635.47} C_VEL
LIN {X 0,Y 503.957,Z 537.713,A -85,B 0,C 180,E1 -5636.334,E2 -5636.334} C_VEL
LIN {X 0,Y 502.91,Z 537.84,A -85,B 0,C 180,E1 -5637,E2 -5637} C_VEL
LIN {X 0,Y 502.812,Z 537.85,A -85,B 0,C 180,E1 -5637.225,E2 -5637.225} C_VEL
LIN {X 0,Y 502.818,Z 537.856,A -85,B 0,C 180,E1 -5640.065,E2 -5640.065} C_VEL
LIN {X 0,Y 502.856,Z 537.904,A -85,B 0,C 180,E1 -5642.635,E2 -5642.635} C_VEL
LIN {X 0,Y 505.461,Z 550.203,A -85,B 0,C 180,E1 -5644.467,E2 -5644.467} C_VEL
LIN {X 0,Y 505.443,Z 558.017,A -85,B 0,C 180,E1 -5645.565,E2 -5645.565} C_VEL
LIN {X 0,Y 504.761,Z 579.532,A -85,B 0,C 180,E1 -5648.562,E2 -5648.562} C_VEL
LIN {X 0,Y 504.208,Z 601.31,A -85,B 0,C 180,E1 -5651.549,E2 -5651.549} C_VEL
LIN {X 0,Y 503.787,Z 621.464,A -85,B 0,C 180,E1 -5654.241,E2 -5654.241} C_VEL
LIN {X 0,Y 505.414,Z 632.847,A -85,B 0,C 180,E1 -5654.463,E2 -5654.463} C_VEL
LIN {X 0,Y 504.929,Z 730.451,A -85,B 0,C 180,E1 -5655.876,E2 -5655.876} C_VEL
LIN {X 0,Y 504.689,Z 743.147,A -85,B 0,C 180,E1 -5656.203,E2 -5656.203} C_VEL
LIN {X 0,Y 504.364,Z 756.037,A -85,B 0,C 180,E1 -5656.707,E2 -5656.707} C_VEL
LIN {X 0,Y 504.051,Z 768.224,A -85,B 0,C 180,E1 -5657.363,E2 -5657.363} C_VEL
LIN {X 0,Y 503.732,Z 779.233,A -85,B 0,C 180,E1 -5658.124,E2 -5658.124} C_VEL
LIN {X 0,Y 503.322,Z 789.683,A -85,B 0,C 180,E1 -5659.032,E2 -5659.032} C_VEL
LIN {X 0,Y 502.972,Z 799.965,A -85,B 0,C 180,E1 -5660.144,E2 -5660.144} C_VEL
LIN {X 0,Y 502.683,Z 808.885,A -85,B 0,C 180,E1 -5661.355,E2 -5661.355} C_VEL
LIN {X 0,Y 502.426,Z 816.057,A -85,B 0,C 180,E1 -5662.565,E2 -5662.565} C_VEL
LIN {X 0,Y 502.343,Z 822.645,A -85,B 0,C 180,E1 -5663.976,E2 -5663.976} C_VEL
LIN {X 0,Y 502.112,Z 826.974,A -85,B 0,C 180,E1 -5665.182,E2 -5665.182} C_VEL
LIN {X 0,Y 502.231,Z 829.246,A -85,B 0,C 180,E1 -5665.987,E2 -5665.987} C_VEL
LIN {X 0,Y 502.124,Z 831.105,A -85,B 0,C 180,E1 -5666.79,E2 -5666.79} C_VEL
LIN {X 0,Y 502.121,Z 832.529,A -85,B 0,C 180,E1 -5667.593,E2 -5667.593} C_VEL
LIN {X 0,Y 501.991,Z 834.145,A -85,B 0,C 180,E1 -5669.197,E2 -5669.197} C_VEL
LIN {X 0,Y 501.98,Z 834.384,A -85,B 0,C 180,E1 -5669.999,E2 -5669.999} C_VEL
LIN {X 0,Y 501.99,Z 834.199,A -85,B 0,C 180,E1 -5670.802,E2 -5670.802} C_VEL
LIN {X 0,Y 502.121,Z 832.655,A -85,B 0,C 180,E1 -5672.406,E2 -5672.406} C_VEL
LIN {X 0,Y 502.124,Z 831.3,A -85,B 0,C 180,E1 -5673.209,E2 -5673.209} C_VEL
LIN {X 0,Y 502.178,Z 828.445,A -85,B 0,C 180,E1 -5674.414,E2 -5674.414} C_VEL
LIN {X 0,Y 502.277,Z 824.563,A -85,B 0,C 180,E1 -5675.62,E2 -5675.62} C_VEL
LIN {X 0,Y 502.342,Z 819.545,A -85,B 0,C 180,E1 -5676.829,E2 -5676.829} C_VEL
LIN {X 0,Y 502.545,Z 813.21,A -85,B 0,C 180,E1 -5678.038,E2 -5678.038} C_VEL
LIN {X 0,Y 502.755,Z 805.335,A -85,B 0,C 180,E1 -5679.25,E2 -5679.25} C_VEL
LIN {X 0,Y 503.03,Z 797.289,A -85,B 0,C 180,E1 -5680.26,E2 -5680.26} C_VEL
LIN {X 0,Y 503.45,Z 787.434,A -85,B 0,C 180,E1 -5681.269,E2 -5681.269} C_VEL
LIN {X 0,Y 503.78,Z 776.321,A -85,B 0,C 180,E1 -5682.184,E2 -5682.184} C_VEL
LIN {X 0,Y 504.13,Z 765.566,A -85,B 0,C 180,E1 -5682.888,E2 -5682.888} C_VEL
LIN {X 0,Y 504.461,Z 753.533,A -85,B 0,C 180,E1 -5683.494,E2 -5683.494} C_VEL
LIN {X 0,Y 504.735,Z 740.317,A -85,B 0,C 180,E1 -5683.974,E2 -5683.974} C_VEL
LIN {X 0,Y 504.926,Z 727.181,A -85,B 0,C 180,E1 -5684.277,E2 -5684.277} C_VEL
LIN {X 0,Y 505.358,Z 633.213,A -85,B 0,C 180,E1 -5685.623,E2 -5685.623} C_VEL
LIN {X 0,Y 503.514,Z 621.959,A -85,B 0,C 180,E1 -5685.863,E2 -5685.863} C_VEL
LIN {X 0,Y 504.015,Z 601.69,A -85,B 0,C 180,E1 -5688.916,E2 -5688.916} C_VEL
LIN {X 0,Y 504.483,Z 583.791,A -85,B 0,C 180,E1 -5691.664,E2 -5691.664} C_VEL
LIN {X 0,Y 505.012,Z 564.539,A -85,B 0,C 180,E1 -5694.675,E2 -5694.675} C_VEL
LIN {X 0,Y 505.391,Z 551.132,A -85,B 0,C 180,E1 -5696.784,E2 -5696.784} C_VEL
LIN {X 0,Y 503.659,Z 541.778,A -85,B 0,C 180,E1 -5698.321,E2 -5698.321} C_VEL
LIN {X 0,Y 502.845,Z 537.852,A -85,B 0,C 180,E1 -5698.998,E2 -5698.998} C_VEL
LIN {X 0,Y 502.786,Z 537.854,A -85,B 0,C 180,E1 -5702.083,E2 -5702.083} C_VEL
LIN {X 0,Y 502.808,Z 537.856,A -85,B 0,C 180,E1 -5704.964,E2 -5704.964} C_VEL
LIN {X 0,Y 502.792,Z 537.854,A -85,B 0,C 180,E1 -5707.952,E2 -5707.952} C_VEL
LIN {X 0,Y 502.816,Z 537.853,A -85,B 0,C 180,E1 -5711.065,E2 -5711.065} C_VEL
LIN {X 0,Y 502.784,Z 537.848,A -85,B 0,C 180,E1 -5714.338,E2 -5714.338} C_VEL
LIN {X 0,Y 502.781,Z 537.854,A -85,B 0,C 180,E1 -5716.769,E2 -5716.769} C_VEL
LIN {X 0,Y 502.822,Z 537.851,A -85,B 0,C 180,E1 -5719.003,E2 -5719.003} C_VEL
LIN {X 0,Y 502.803,Z 537.853,A -85,B 0,C 180,E1 -5722.047,E2 -5722.047} C_VEL
LIN {X 0,Y 502.865,Z 538.041,A -85,B 0,C 180,E1 -5722.702,E2 -5722.702} C_VEL
LIN {X 0,Y 505.369,Z 545.603,A -85,B 0,C 180,E1 -5722.897,E2 -5722.897} C_VEL
LIN {X 0,Y 504.84,Z 618.09,A -85,B 0,C 180,E1 -5723.99,E2 -5723.99} C_VEL
LIN {X 0,Y 504.766,Z 631.065,A -85,B 0,C 180,E1 -5724.351,E2 -5724.351} C_VEL
LIN {X 0,Y 504.614,Z 643.861,A -85,B 0,C 180,E1 -5724.874,E2 -5724.874} C_VEL
LIN {X 0,Y 504.352,Z 655.52,A -85,B 0,C 180,E1 -5725.521,E2 -5725.521} C_VEL
LIN {X 0,Y 504.066,Z 666.577,A -85,B 0,C 180,E1 -5726.306,E2 -5726.306} C_VEL
LIN {X 0,Y 503.77,Z 677.466,A -85,B 0,C 180,E1 -5727.276,E2 -5727.276} C_VEL
LIN {X 0,Y 503.432,Z 687.322,A -85,B 0,C 180,E1 -5728.38,E2 -5728.38} C_VEL
LIN {X 0,Y 503.187,Z 695.965,A -85,B 0,C 180,E1 -5729.582,E2 -5729.582} C_VEL
LIN {X 0,Y 502.944,Z 702.564,A -85,B 0,C 180,E1 -5730.72,E2 -5730.72} C_VEL
LIN {X 0,Y 502.735,Z 708.955,A -85,B 0,C 180,E1 -5732.12,E2 -5732.12} C_VEL
LIN {X 0,Y 502.668,Z 713.669,A -85,B 0,C 180,E1 -5733.481,E2 -5733.481} C_VEL
LIN {X 0,Y 502.581,Z 715.895,A -85,B 0,C 180,E1 -5734.31,E2 -5734.31} C_VEL
LIN {X 0,Y 502.486,Z 718.076,A -85,B 0,C 180,E1 -5735.38,E2 -5735.38} C_VEL
LIN {X 0,Y 502.488,Z 719.095,A -85,B 0,C 180,E1 -5736.071,E2 -5736.071} C_VEL
LIN {X 0,Y 502.474,Z 720.213,A -85,B 0,C 180,E1 -5737.384,E2 -5737.384} C_VEL
LIN {X 0,Y 502.46,Z 720.285,A -85,B 0,C 180,E1 -5738.674,E2 -5738.674} C_VEL
LIN {X 0,Y 502.469,Z 719.711,A -85,B 0,C 180,E1 -5739.57,E2 -5739.57} C_VEL
LIN {X 0,Y 502.512,Z 718.78,A -85,B 0,C 180,E1 -5740.387,E2 -5740.387} C_VEL
LIN {X 0,Y 502.594,Z 717.371,A -85,B 0,C 180,E1 -5741.239,E2 -5741.239} C_VEL
LIN {X 0,Y 502.712,Z 714.354,A -85,B 0,C 180,E1 -5742.508,E2 -5742.508} C_VEL
LIN {X 0,Y 502.808,Z 710.237,A -85,B 0,C 180,E1 -5743.767,E2 -5743.767} C_VEL
LIN {X 0,Y 503.045,Z 703.846,A -85,B 0,C 180,E1 -5745.233,E2 -5745.233} C_VEL
LIN {X 0,Y 503.272,Z 696.894,A -85,B 0,C 180,E1 -5746.473,E2 -5746.473} C_VEL
LIN {X 0,Y 503.526,Z 688.297,A -85,B 0,C 180,E1 -5747.688,E2 -5747.688} C_VEL
LIN {X 0,Y 503.853,Z 679.08,A -85,B 0,C 180,E1 -5748.739,E2 -5748.739} C_VEL
LIN {X 0,Y 504.17,Z 669.06,A -85,B 0,C 180,E1 -5749.661,E2 -5749.661} C_VEL
LIN {X 0,Y 504.44,Z 657.928,A -85,B 0,C 180,E1 -5750.477,E2 -5750.477} C_VEL
LIN {X 0,Y 504.693,Z 647.353,A -85,B 0,C 180,E1 -5751.088,E2 -5751.088} C_VEL
LIN {X 0,Y 504.816,Z 635.267,A -85,B 0,C 180,E1 -5751.624,E2 -5751.624} C_VEL
LIN {X 0,Y 504.868,Z 622.394,A -85,B 0,C 180,E1 -5752.018,E2 -5752.018} C_VEL
LIN {X 0,Y 504.915,Z 605.157,A -85,B 0,C 180,E1 -5752.32,E2 -5752.32} C_VEL
LIN {X 0,Y 505.236,Z 545.013,A -85,B 0,C 180,E1 -5753.225,E2 -5753.225} C_VEL
LIN {X 0,Y 502.904,Z 537.841,A -85,B 0,C 180,E1 -5753.428,E2 -5753.428} C_VEL
LIN {X 0,Y 502.873,Z 537.845,A -85,B 0,C 180,E1 -5755.19,E2 -5755.19} C_VEL
LIN {X 0,Y 503.018,Z 537.824,A -85,B 0,C 180,E1 -5757.598,E2 -5757.598} C_VEL
LIN {X 0,Y 503.016,Z 537.826,A -85,B 0,C 180,E1 -5760,E2 -5760} C_VEL
LIN {X 0,Y 503.015,Z 537.829,A -85,B 0,C 180,E1 -5762.402,E2 -5762.402} C_VEL
LIN {X 0,Y 502.952,Z 537.831,A -85,B 0,C 180,E1 -5765.613,E2 -5765.613} C_VEL
LIN {X 0,Y 502.891,Z 537.838,A -85,B 0,C 180,E1 -5768.033,E2 -5768.033} C_VEL
LIN {X 0,Y 502.884,Z 537.842,A -85,B 0,C 180,E1 -5771.283,E2 -5771.283} C_VEL
LIN {X 0,Y 502.84,Z 537.851,A -85,B 0,C 180,E1 -5774.571,E2 -5774.571} C_VEL
LIN {X 0,Y 502.851,Z 537.844,A -85,B 0,C 180,E1 -5777.907,E2 -5777.907} C_VEL
LIN {X 0,Y 502.818,Z 537.853,A -85,B 0,C 180,E1 -5780.537,E2 -5780.537} C_VEL
LIN {X 0,Y 502.787,Z 537.857,A -85,B 0,C 180,E1 -5783.041,E2 -5783.041} C_VEL
LIN {X 0,Y 502.832,Z 537.845,A -85,B 0,C 180,E1 -5785.676,E2 -5785.676} C_VEL
LIN {X 0,Y 502.833,Z 537.848,A -85,B 0,C 180,E1 -5788.373,E2 -5788.373} C_VEL
LIN {X 0,Y 502.788,Z 537.852,A -85,B 0,C 180,E1 -5791.5,E2 -5791.5} C_VEL
LIN {X 0,Y 502.799,Z 537.854,A -85,B 0,C 180,E1 -5794.446,E2 -5794.446} C_VEL
LIN {X 0,Y 502.774,Z 537.855,A -85,B 0,C 180,E1 -5797.179,E2 -5797.179} C_VEL
LIN {X 0,Y 502.82,Z 537.847,A -85,B 0,C 180,E1 -5800.012,E2 -5800.012} C_VEL
LIN {X 0,Y 502.82,Z 537.85,A -85,B 0,C 180,E1 -5802.203,E2 -5802.203} C_VEL
LIN {X 0,Y 502.794,Z 537.853,A -85,B 0,C 180,E1 -5805.469,E2 -5805.469} C_VEL
LIN {X 0,Y 502.824,Z 537.848,A -85,B 0,C 180,E1 -5807.865,E2 -5807.865} C_VEL
LIN {X 0,Y 502.818,Z 537.856,A -85,B 0,C 180,E1 -5811.027,E2 -5811.027} C_VEL
LIN {X 0,Y 502.783,Z 537.856,A -85,B 0,C 180,E1 -5814.168,E2 -5814.168} C_VEL
LIN {X 0,Y 502.83,Z 537.854,A -85,B 0,C 180,E1 -5816.994,E2 -5816.994} C_VEL
LIN {X 0,Y 502.812,Z 537.853,A -85,B 0,C 180,E1 -5820.066,E2 -5820.066} C_VEL
LIN {X 0,Y 502.867,Z 538.018,A -85,B 0,C 180,E1 -5820.879,E2 -5820.879} C_VEL
LIN {X 0,Y 505.819,Z 551.662,A -85,B 0,C 180,E1 -5822.778,E2 -5822.778} C_VEL
LIN {X 0,Y 505.338,Z 570.635,A -85,B 0,C 180,E1 -5825.159,E2 -5825.159} C_VEL
LIN {X 0,Y 504.738,Z 593.159,A -85,B 0,C 180,E1 -5827.918,E2 -5827.918} C_VEL
LIN {X 0,Y 504.115,Z 619.52,A -85,B 0,C 180,E1 -5831.088,E2 -5831.088} C_VEL
LIN {X 0,Y 503.534,Z 645.369,A -85,B 0,C 180,E1 -5834.166,E2 -5834.166} C_VEL
LIN {X 0,Y 505.285,Z 662.508,A -85,B 0,C 180,E1 -5834.492,E2 -5834.492} C_VEL
LIN {X 0,Y 504.732,Z 756.656,A -85,B 0,C 180,E1 -5835.872,E2 -5835.872} C_VEL
LIN {X 0,Y 504.397,Z 770.665,A -85,B 0,C 180,E1 -5836.248,E2 -5836.248} C_VEL
LIN {X 0,Y 504.129,Z 783.265,A -85,B 0,C 180,E1 -5836.754,E2 -5836.754} C_VEL
LIN {X 0,Y 503.826,Z 794.632,A -85,B 0,C 180,E1 -5837.364,E2 -5837.364} C_VEL
LIN {X 0,Y 503.511,Z 805.771,A -85,B 0,C 180,E1 -5838.12,E2 -5838.12} C_VEL
LIN {X 0,Y 503.171,Z 816.501,A -85,B 0,C 180,E1 -5839.03,E2 -5839.03} C_VEL
LIN {X 0,Y 502.88,Z 825.266,A -85,B 0,C 180,E1 -5839.94,E2 -5839.94} C_VEL
LIN {X 0,Y 502.661,Z 833.377,A -85,B 0,C 180,E1 -5840.951,E2 -5840.951} C_VEL
LIN {X 0,Y 502.487,Z 840.143,A -85,B 0,C 180,E1 -5841.961,E2 -5841.961} C_VEL
LIN {X 0,Y 502.354,Z 845.879,A -85,B 0,C 180,E1 -5842.99,E2 -5842.99} C_VEL
LIN {X 0,Y 502.306,Z 850.489,A -85,B 0,C 180,E1 -5843.977,E2 -5843.977} C_VEL
LIN {X 0,Y 502.167,Z 854.956,A -85,B 0,C 180,E1 -5845.184,E2 -5845.184} C_VEL
LIN {X 0,Y 502.25,Z 857.374,A -85,B 0,C 180,E1 -5845.989,E2 -5845.989} C_VEL
LIN {X 0,Y 502.148,Z 860.725,A -85,B 0,C 180,E1 -5847.594,E2 -5847.594} C_VEL
LIN {X 0,Y 502.078,Z 861.764,A -85,B 0,C 180,E1 -5848.396,E2 -5848.396} C_VEL
LIN {X 0,Y 502.061,Z 862.612,A -85,B 0,C 180,E1 -5850.001,E2 -5850.001} C_VEL
LIN {X 0,Y 502.076,Z 861.783,A -85,B 0,C 180,E1 -5851.605,E2 -5851.605} C_VEL
LIN {X 0,Y 502.143,Z 860.772,A -85,B 0,C 180,E1 -5852.407,E2 -5852.407} C_VEL
LIN {X 0,Y 502.155,Z 859.326,A -85,B 0,C 180,E1 -5853.21,E2 -5853.21} C_VEL
LIN {X 0,Y 502.183,Z 856.317,A -85,B 0,C 180,E1 -5854.415,E2 -5854.415} C_VEL
LIN {X 0,Y 502.281,Z 852.243,A -85,B 0,C 180,E1 -5855.621,E2 -5855.621} C_VEL
LIN {X 0,Y 502.337,Z 846.086,A -85,B 0,C 180,E1 -5857.012,E2 -5857.012} C_VEL
LIN {X 0,Y 502.505,Z 839.141,A -85,B 0,C 180,E1 -5858.243,E2 -5858.243} C_VEL
LIN {X 0,Y 502.731,Z 830.585,A -85,B 0,C 180,E1 -5859.455,E2 -5859.455} C_VEL
LIN {X 0,Y 502.964,Z 821.891,A -85,B 0,C 180,E1 -5860.466,E2 -5860.466} C_VEL
LIN {X 0,Y 503.329,Z 811.239,A -85,B 0,C 180,E1 -5861.477,E2 -5861.477} C_VEL
LIN {X 0,Y 503.604,Z 799.806,A -85,B 0,C 180,E1 -5862.344,E2 -5862.344} C_VEL
LIN {X 0,Y 503.981,Z 788.96,A -85,B 0,C 180,E1 -5862.995,E2 -5862.995} C_VEL
LIN {X 0,Y 504.331,Z 776.952,A -85,B 0,C 180,E1 -5863.55,E2 -5863.55} C_VEL
LIN {X 0,Y 504.615,Z 763.963,A -85,B 0,C 180,E1 -5863.979,E2 -5863.979} C_VEL
LIN {X 0,Y 504.813,Z 750.39,A -85,B 0,C 180,E1 -5864.256,E2 -5864.256} C_VEL
LIN {X 0,Y 505.234,Z 661.446,A -85,B 0,C 180,E1 -5865.539,E2 -5865.539} C_VEL
LIN {X 0,Y 503.444,Z 647.282,A -85,B 0,C 180,E1 -5865.824,E2 -5865.824} C_VEL
LIN {X 0,Y 503.979,Z 622.717,A -85,B 0,C 180,E1 -5869.13,E2 -5869.13} C_VEL
LIN {X 0,Y 504.559,Z 601.04,A -85,B 0,C 180,E1 -5872.092,E2 -5872.092} C_VEL
LIN {X 0,Y 505.299,Z 577.881,A -85,B 0,C 180,E1 -5875.303,E2 -5875.303} C_VEL
LIN {X 0,Y 506.034,Z 554.598,A -85,B 0,C 180,E1 -5878.602,E2 -5878.602} C_VEL
LIN {X 0,Y 505.793,Z 551.245,A -85,B 0,C 180,E1 -5879.1,E2 -5879.1} C_VEL
LIN {X 0,Y 502.812,Z 537.856,A -85,B 0,C 180,E1 -5881.231,E2 -5881.231} C_VEL
LIN {X 0,Y 502.809,Z 537.85,A -85,B 0,C 180,E1 -5883.994,E2 -5883.994} C_VEL
LIN {X 0,Y 502.78,Z 537.859,A -85,B 0,C 180,E1 -5887.178,E2 -5887.178} C_VEL
LIN {X 0,Y 502.79,Z 537.851,A -85,B 0,C 180,E1 -5890.015,E2 -5890.015} C_VEL
LIN {X 0,Y 502.805,Z 537.849,A -85,B 0,C 180,E1 -5892.199,E2 -5892.199} C_VEL
LIN {X 0,Y 502.803,Z 537.854,A -85,B 0,C 180,E1 -5895.468,E2 -5895.468} C_VEL
LIN {X 0,Y 502.832,Z 537.842,A -85,B 0,C 180,E1 -5897.864,E2 -5897.864} C_VEL
LIN {X 0,Y 502.804,Z 537.855,A -85,B 0,C 180,E1 -5901.024,E2 -5901.024} C_VEL
LIN {X 0,Y 502.786,Z 537.848,A -85,B 0,C 180,E1 -5904.167,E2 -5904.167} C_VEL
LIN {X 0,Y 502.833,Z 537.85,A -85,B 0,C 180,E1 -5906.993,E2 -5906.993} C_VEL
LIN {X 0,Y 502.815,Z 537.846,A -85,B 0,C 180,E1 -5910.065,E2 -5910.065} C_VEL
LIN {X 0,Y 502.834,Z 537.845,A -85,B 0,C 180,E1 -5912.533,E2 -5912.533} C_VEL
LIN {X 0,Y 502.827,Z 537.846,A -85,B 0,C 180,E1 -5915.299,E2 -5915.299} C_VEL
LIN {X 0,Y 502.78,Z 537.855,A -85,B 0,C 180,E1 -5917.826,E2 -5917.826} C_VEL
LIN {X 0,Y 502.825,Z 537.844,A -85,B 0,C 180,E1 -5920.4,E2 -5920.4} C_VEL
LIN {X 0,Y 502.834,Z 537.839,A -85,B 0,C 180,E1 -5922.932,E2 -5922.932} C_VEL
LIN {X 0,Y 502.851,Z 537.85,A -85,B 0,C 180,E1 -5925.429,E2 -5925.429} C_VEL
LIN {X 0,Y 502.877,Z 537.835,A -85,B 0,C 180,E1 -5928.717,E2 -5928.717} C_VEL
LIN {X 0,Y 502.901,Z 537.84,A -85,B 0,C 180,E1 -5931.967,E2 -5931.967} C_VEL
LIN {X 0,Y 502.938,Z 537.832,A -85,B 0,C 180,E1 -5934.387,E2 -5934.387} C_VEL
LIN {X 0,Y 503.024,Z 537.82,A -85,B 0,C 180,E1 -5937.598,E2 -5937.598} C_VEL
LIN {X 0,Y 503.026,Z 537.825,A -85,B 0,C 180,E1 -5940,E2 -5940} C_VEL
LIN {X 0,Y 503.024,Z 537.821,A -85,B 0,C 180,E1 -5942.402,E2 -5942.402} C_VEL
LIN {X 0,Y 502.938,Z 537.829,A -85,B 0,C 180,E1 -5945.614,E2 -5945.614} C_VEL
LIN {X 0,Y 502.902,Z 537.842,A -85,B 0,C 180,E1 -5948.033,E2 -5948.033} C_VEL
LIN {X 0,Y 502.877,Z 537.839,A -85,B 0,C 180,E1 -5951.283,E2 -5951.283} C_VEL
LIN {X 0,Y 502.845,Z 537.844,A -85,B 0,C 180,E1 -5954.571,E2 -5954.571} C_VEL
LIN {X 0,Y 502.862,Z 537.845,A -85,B 0,C 180,E1 -5957.907,E2 -5957.907} C_VEL
LIN {X 0,Y 502.829,Z 537.846,A -85,B 0,C 180,E1 -5960.536,E2 -5960.536} C_VEL
LIN {X 0,Y 502.795,Z 537.85,A -85,B 0,C 180,E1 -5963.041,E2 -5963.041} C_VEL
LIN {X 0,Y 502.841,Z 537.843,A -85,B 0,C 180,E1 -5965.676,E2 -5965.676} C_VEL
LIN {X 0,Y 502.841,Z 537.848,A -85,B 0,C 180,E1 -5968.373,E2 -5968.373} C_VEL
LIN {X 0,Y 502.793,Z 537.848,A -85,B 0,C 180,E1 -5971.499,E2 -5971.499} C_VEL
LIN {X 0,Y 502.805,Z 537.857,A -85,B 0,C 180,E1 -5973.994,E2 -5973.994} C_VEL
LIN {X 0,Y 502.779,Z 537.853,A -85,B 0,C 180,E1 -5977.178,E2 -5977.178} C_VEL
LIN {X 0,Y 502.79,Z 537.855,A -85,B 0,C 180,E1 -5980.015,E2 -5980.015} C_VEL
LIN {X 0,Y 502.805,Z 537.856,A -85,B 0,C 180,E1 -5982.199,E2 -5982.199} C_VEL
LIN {X 0,Y 502.787,Z 537.852,A -85,B 0,C 180,E1 -5985.47,E2 -5985.47} C_VEL
LIN {X 0,Y 502.822,Z 537.849,A -85,B 0,C 180,E1 -5988.934,E2 -5988.934} C_VEL
LIN {X 0,Y 502.795,Z 537.851,A -85,B 0,C 180,E1 -5992.046,E2 -5992.046} C_VEL
LIN {X 0,Y 502.807,Z 537.851,A -85,B 0,C 180,E1 -5995.035,E2 -5995.035} C_VEL
LIN {X 0,Y 502.812,Z 537.85,A -85,B 0,C 180,E1 -5997.225,E2 -5997.225} C_VEL
LIN {X 0,Y 502.111,Z 537.94,A -85,B 0,C 180,E1 -5997.894,E2 -5997.894} C_VEL
LIN {X 0,Y 499.246,Z 538.3,A -85,B 0,C 180,E1 -5998.98,E2 -5998.98} C_VEL
LIN {X 0,Y 496.852,Z 538.599,A -85,B 0,C 180,E1 -5999.855,E2 -5999.855} C_VEL
LIN {X 0,Y 495.835,Z 538.727,A -85,B 0,C 180,E1 -6000.53,E2 -6000.53} C_VEL
LIN {X 0,Y 495.757,Z 538.733,A -85,B 0,C 180,E1 -6000.759,E2 -6000.759} C_VEL
LIN {X 0,Y 495.847,Z 538.891,A -85,B 0,C 180,E1 -6002.428,E2 -6002.428} C_VEL
LIN {X 0,Y 498.652,Z 552.139,A -85,B 0,C 180,E1 -6004.425,E2 -6004.425} C_VEL
LIN {X 0,Y 498.319,Z 566.518,A -85,B 0,C 180,E1 -6006.452,E2 -6006.452} C_VEL
LIN {X 0,Y 497.581,Z 588.436,A -85,B 0,C 180,E1 -6009.538,E2 -6009.538} C_VEL
LIN {X 0,Y 497.025,Z 610.208,A -85,B 0,C 180,E1 -6012.513,E2 -6012.513} C_VEL
LIN {X 0,Y 496.846,Z 621.4,A -85,B 0,C 180,E1 -6014.004,E2 -6014.004} C_VEL
LIN {X 0,Y 498.613,Z 634.621,A -85,B 0,C 180,E1 -6014.27,E2 -6014.27} C_VEL
LIN {X 0,Y 498.059,Z 730.542,A -85,B 0,C 180,E1 -6015.677,E2 -6015.677} C_VEL
LIN {X 0,Y 497.821,Z 743.282,A -85,B 0,C 180,E1 -6016.009,E2 -6016.009} C_VEL
LIN {X 0,Y 497.453,Z 756.197,A -85,B 0,C 180,E1 -6016.519,E2 -6016.519} C_VEL
LIN {X 0,Y 497.102,Z 768.856,A -85,B 0,C 180,E1 -6017.212,E2 -6017.212} C_VEL
LIN {X 0,Y 496.79,Z 779.411,A -85,B 0,C 180,E1 -6017.955,E2 -6017.955} C_VEL
LIN {X 0,Y 496.331,Z 789.867,A -85,B 0,C 180,E1 -6018.876,E2 -6018.876} C_VEL
LIN {X 0,Y 495.982,Z 800.152,A -85,B 0,C 180,E1 -6020.003,E2 -6020.003} C_VEL
LIN {X 0,Y 495.644,Z 809.076,A -85,B 0,C 180,E1 -6021.232,E2 -6021.232} C_VEL
LIN {X 0,Y 495.369,Z 816.249,A -85,B 0,C 180,E1 -6022.459,E2 -6022.459} C_VEL
LIN {X 0,Y 495.281,Z 822.837,A -85,B 0,C 180,E1 -6023.89,E2 -6023.89} C_VEL
LIN {X 0,Y 495.04,Z 827.168,A -85,B 0,C 180,E1 -6025.113,E2 -6025.113} C_VEL
LIN {X 0,Y 495.142,Z 829.44,A -85,B 0,C 180,E1 -6025.93,E2 -6025.93} C_VEL
LIN {X 0,Y 495.05,Z 831.299,A -85,B 0,C 180,E1 -6026.744,E2 -6026.744} C_VEL
LIN {X 0,Y 495.024,Z 832.723,A -85,B 0,C 180,E1 -6027.558,E2 -6027.558} C_VEL
LIN {X 0,Y 494.911,Z 834.338,A -85,B 0,C 180,E1 -6029.186,E2 -6029.186} C_VEL
LIN {X 0,Y 494.898,Z 834.576,A -85,B 0,C 180,E1 -6029.999,E2 -6029.999} C_VEL
LIN {X 0,Y 494.911,Z 834.391,A -85,B 0,C 180,E1 -6030.813,E2 -6030.813} C_VEL
LIN {X 0,Y 495.025,Z 832.847,A -85,B 0,C 180,E1 -6032.44,E2 -6032.44} C_VEL
LIN {X 0,Y 495.05,Z 831.491,A -85,B 0,C 180,E1 -6033.255,E2 -6033.255} C_VEL
LIN {X 0,Y 495.093,Z 828.635,A -85,B 0,C 180,E1 -6034.477,E2 -6034.477} C_VEL
LIN {X 0,Y 495.233,Z 823.602,A -85,B 0,C 180,E1 -6036.002,E2 -6036.002} C_VEL
LIN {X 0,Y 495.341,Z 817.77,A -85,B 0,C 180,E1 -6037.336,E2 -6037.336} C_VEL
LIN {X 0,Y 495.578,Z 810.98,A -85,B 0,C 180,E1 -6038.563,E2 -6038.563} C_VEL
LIN {X 0,Y 495.874,Z 802.467,A -85,B 0,C 180,E1 -6039.791,E2 -6039.791} C_VEL
LIN {X 0,Y 496.215,Z 793.76,A -85,B 0,C 180,E1 -6040.816,E2 -6040.816} C_VEL
LIN {X 0,Y 496.63,Z 784.215,A -85,B 0,C 180,E1 -6041.737,E2 -6041.737} C_VEL
LIN {X 0,Y 496.933,Z 773.431,A -85,B 0,C 180,E1 -6042.576,E2 -6042.576} C_VEL
LIN {X 0,Y 497.304,Z 762.033,A -85,B 0,C 180,E1 -6043.275,E2 -6043.275} C_VEL
LIN {X 0,Y 497.643,Z 750.039,A -85,B 0,C 180,E1 -6043.838,E2 -6043.838} C_VEL
LIN {X 0,Y 497.926,Z 737.693,A -85,B 0,C 180,E1 -6044.247,E2 -6044.247} C_VEL
LIN {X 0,Y 498.113,Z 723.824,A -85,B 0,C 180,E1 -6044.529,E2 -6044.529} C_VEL
LIN {X 0,Y 498.5,Z 633.758,A -85,B 0,C 180,E1 -6045.836,E2 -6045.836} C_VEL
LIN {X 0,Y 496.591,Z 622.215,A -85,B 0,C 180,E1 -6046.078,E2 -6046.078} C_VEL
LIN {X 0,Y 497.05,Z 601.492,A -85,B 0,C 180,E1 -6049.191,E2 -6049.191} C_VEL
LIN {X 0,Y 497.54,Z 583.515,A -85,B 0,C 180,E1 -6051.982,E2 -6051.982} C_VEL
LIN {X 0,Y 498.11,Z 565.616,A -85,B 0,C 180,E1 -6054.818,E2 -6054.818} C_VEL
LIN {X 0,Y 498.512,Z 553.018,A -85,B 0,C 180,E1 -6056.815,E2 -6056.815} C_VEL
LIN {X 0,Y 497.288,Z 545.756,A -85,B 0,C 180,E1 -6058.019,E2 -6058.019} C_VEL
LIN {X 0,Y 495.785,Z 538.732,A -85,B 0,C 180,E1 -6059.219,E2 -6059.219} C_VEL
LIN {X 0,Y 495.767,Z 538.729,A -85,B 0,C 180,E1 -6062.593,E2 -6062.593} C_VEL
LIN {X 0,Y 495.755,Z 538.731,A -85,B 0,C 180,E1 -6065.536,E2 -6065.536} C_VEL
LIN {X 0,Y 495.761,Z 538.732,A -85,B 0,C 180,E1 -6068.767,E2 -6068.767} C_VEL
LIN {X 0,Y 495.772,Z 538.727,A -85,B 0,C 180,E1 -6071.778,E2 -6071.778} C_VEL
LIN {X 0,Y 495.744,Z 538.731,A -85,B 0,C 180,E1 -6075.138,E2 -6075.138} C_VEL
LIN {X 0,Y 495.779,Z 538.725,A -85,B 0,C 180,E1 -6078.221,E2 -6078.221} C_VEL
LIN {X 0,Y 495.772,Z 538.733,A -85,B 0,C 180,E1 -6081.228,E2 -6081.228} C_VEL
LIN {X 0,Y 495.764,Z 538.729,A -85,B 0,C 180,E1 -6082.471,E2 -6082.471} C_VEL
LIN {X 0,Y 498.526,Z 547.61,A -85,B 0,C 180,E1 -6082.713,E2 -6082.713} C_VEL
LIN {X 0,Y 497.957,Z 618.695,A -85,B 0,C 180,E1 -6083.802,E2 -6083.802} C_VEL
LIN {X 0,Y 497.89,Z 631.871,A -85,B 0,C 180,E1 -6084.172,E2 -6084.172} C_VEL
LIN {X 0,Y 497.744,Z 644.38,A -85,B 0,C 180,E1 -6084.687,E2 -6084.687} C_VEL
LIN {X 0,Y 497.492,Z 655.564,A -85,B 0,C 180,E1 -6085.305,E2 -6085.305} C_VEL
LIN {X 0,Y 497.187,Z 666.256,A -85,B 0,C 180,E1 -6086.058,E2 -6086.058} C_VEL
LIN {X 0,Y 496.861,Z 677.024,A -85,B 0,C 180,E1 -6087.004,E2 -6087.004} C_VEL
LIN {X 0,Y 496.556,Z 686.636,A -85,B 0,C 180,E1 -6088.053,E2 -6088.053} C_VEL
LIN {X 0,Y 496.294,Z 694.533,A -85,B 0,C 180,E1 -6089.114,E2 -6089.114} C_VEL
LIN {X 0,Y 496.011,Z 701.593,A -85,B 0,C 180,E1 -6090.27,E2 -6090.27} C_VEL
LIN {X 0,Y 495.809,Z 707.649,A -85,B 0,C 180,E1 -6091.499,E2 -6091.499} C_VEL
LIN {X 0,Y 495.69,Z 713.411,A -85,B 0,C 180,E1 -6093.018,E2 -6093.018} C_VEL
LIN {X 0,Y 495.557,Z 717.113,A -85,B 0,C 180,E1 -6094.37,E2 -6094.37} C_VEL
LIN {X 0,Y 495.455,Z 719.615,A -85,B 0,C 180,E1 -6095.709,E2 -6095.709} C_VEL
LIN {X 0,Y 495.436,Z 721.126,A -85,B 0,C 180,E1 -6097.225,E2 -6097.225} C_VEL
LIN {X 0,Y 495.445,Z 721.346,A -85,B 0,C 180,E1 -6098.357,E2 -6098.357} C_VEL
LIN {X 0,Y 495.452,Z 720.886,A -85,B 0,C 180,E1 -6099.42,E2 -6099.42} C_VEL
LIN {X 0,Y 495.553,Z 718.958,A -85,B 0,C 180,E1 -6100.962,E2 -6100.962} C_VEL
LIN {X 0,Y 495.664,Z 716.217,A -85,B 0,C 180,E1 -6102.251,E2 -6102.251} C_VEL
LIN {X 0,Y 495.781,Z 712.392,A -85,B 0,C 180,E1 -6103.53,E2 -6103.53} C_VEL
LIN {X 0,Y 495.982,Z 707.11,A -85,B 0,C 180,E1 -6104.864,E2 -6104.864} C_VEL
LIN {X 0,Y 496.235,Z 700.998,A -85,B 0,C 180,E1 -6106.068,E2 -6106.068} C_VEL
LIN {X 0,Y 496.487,Z 692.995,A -85,B 0,C 180,E1 -6107.326,E2 -6107.326} C_VEL
LIN {X 0,Y 496.793,Z 684.793,A -85,B 0,C 180,E1 -6108.37,E2 -6108.37} C_VEL
LIN {X 0,Y 497.082,Z 674.763,A -85,B 0,C 180,E1 -6109.409,E2 -6109.409} C_VEL
LIN {X 0,Y 497.457,Z 663.319,A -85,B 0,C 180,E1 -6110.342,E2 -6110.342} C_VEL
LIN {X 0,Y 497.727,Z 652.093,A -85,B 0,C 180,E1 -6111.064,E2 -6111.064} C_VEL
LIN {X 0,Y 497.896,Z 640.292,A -85,B 0,C 180,E1 -6111.645,E2 -6111.645} C_VEL
LIN {X 0,Y 498.001,Z 626.743,A -85,B 0,C 180,E1 -6112.117,E2 -6112.117} C_VEL
LIN {X 0,Y 498.038,Z 613.628,A -85,B 0,C 180,E1 -6112.398,E2 -6112.398} C_VEL
LIN {X 0,Y 498.523,Z 546.63,A -85,B 0,C 180,E1 -6113.423,E2 -6113.423} C_VEL
LIN {X 0,Y 495.87,Z 538.719,A -85,B 0,C 180,E1 -6113.643,E2 -6113.643} C_VEL
LIN {X 0,Y 495.86,Z 538.722,A -85,B 0,C 180,E1 -6116.75,E2 -6116.75} C_VEL
LIN {X 0,Y 495.996,Z 538.702,A -85,B 0,C 180,E1 -6119.188,E2 -6119.188} C_VEL
LIN {X 0,Y 495.862,Z 538.715,A -85,B 0,C 180,E1 -6121.624,E2 -6121.624} C_VEL
LIN {X 0,Y 495.839,Z 538.72,A -85,B 0,C 180,E1 -6123.25,E2 -6123.25} C_VEL
LIN {X 0,Y 495.872,Z 538.719,A -85,B 0,C 180,E1 -6126.51,E2 -6126.51} C_VEL
LIN {X 0,Y 495.835,Z 538.722,A -85,B 0,C 180,E1 -6128.97,E2 -6128.97} C_VEL
LIN {X 0,Y 495.84,Z 538.72,A -85,B 0,C 180,E1 -6132.275,E2 -6132.275} C_VEL
LIN {X 0,Y 495.796,Z 538.719,A -85,B 0,C 180,E1 -6135.624,E2 -6135.624} C_VEL
LIN {X 0,Y 495.795,Z 538.725,A -85,B 0,C 180,E1 -6138.248,E2 -6138.248} C_VEL
LIN {X 0,Y 495.763,Z 538.734,A -85,B 0,C 180,E1 -6140.757,E2 -6140.757} C_VEL
LIN {X 0,Y 495.742,Z 538.73,A -85,B 0,C 180,E1 -6143.388,E2 -6143.388} C_VEL
LIN {X 0,Y 495.79,Z 538.724,A -85,B 0,C 180,E1 -6146.068,E2 -6146.068} C_VEL
LIN {X 0,Y 495.771,Z 538.732,A -85,B 0,C 180,E1 -6148.815,E2 -6148.815} C_VEL
LIN {X 0,Y 495.75,Z 538.728,A -85,B 0,C 180,E1 -6151.727,E2 -6151.727} C_VEL
LIN {X 0,Y 495.769,Z 538.73,A -85,B 0,C 180,E1 -6154.696,E2 -6154.696} C_VEL
LIN {X 0,Y 495.726,Z 538.73,A -85,B 0,C 180,E1 -6157.562,E2 -6157.562} C_VEL
LIN {X 0,Y 495.787,Z 538.724,A -85,B 0,C 180,E1 -6160.053,E2 -6160.053} C_VEL
LIN {X 0,Y 495.758,Z 538.733,A -85,B 0,C 180,E1 -6162.88,E2 -6162.88} C_VEL
LIN {X 0,Y 495.731,Z 538.732,A -85,B 0,C 180,E1 -6166,E2 -6166} C_VEL
LIN {X 0,Y 495.763,Z 538.734,A -85,B 0,C 180,E1 -6168.706,E2 -6168.706} C_VEL
LIN {X 0,Y 495.76,Z 538.73,A -85,B 0,C 180,E1 -6171.411,E2 -6171.411} C_VEL
LIN {X 0,Y 495.755,Z 538.734,A -85,B 0,C 180,E1 -6174.464,E2 -6174.464} C_VEL
LIN {X 0,Y 495.767,Z 538.731,A -85,B 0,C 180,E1 -6177.407,E2 -6177.407} C_VEL
LIN {X 0,Y 495.811,Z 538.789,A -85,B 0,C 180,E1 -6180.637,E2 -6180.637} C_VEL
LIN {X 0,Y 498.948,Z 553.571,A -85,B 0,C 180,E1 -6182.737,E2 -6182.737} C_VEL
LIN {X 0,Y 498.337,Z 572.87,A -85,B 0,C 180,E1 -6185.194,E2 -6185.194} C_VEL
LIN {X 0,Y 497.649,Z 595.586,A -85,B 0,C 180,E1 -6188.024,E2 -6188.024} C_VEL
LIN {X 0,Y 497.015,Z 621.833,A -85,B 0,C 180,E1 -6191.236,E2 -6191.236} C_VEL
LIN {X 0,Y 496.503,Z 644.285,A -85,B 0,C 180,E1 -6193.948,E2 -6193.948} C_VEL
LIN {X 0,Y 498.403,Z 663.22,A -85,B 0,C 180,E1 -6194.303,E2 -6194.303} C_VEL
LIN {X 0,Y 497.78,Z 756.112,A -85,B 0,C 180,E1 -6195.696,E2 -6195.696} C_VEL
LIN {X 0,Y 497.451,Z 769.936,A -85,B 0,C 180,E1 -6196.078,E2 -6196.078} C_VEL
LIN {X 0,Y 497.129,Z 782.969,A -85,B 0,C 180,E1 -6196.616,E2 -6196.616} C_VEL
LIN {X 0,Y 496.798,Z 794.375,A -85,B 0,C 180,E1 -6197.251,E2 -6197.251} C_VEL
LIN {X 0,Y 496.448,Z 805.869,A -85,B 0,C 180,E1 -6198.052,E2 -6198.052} C_VEL
LIN {X 0,Y 496.102,Z 816.562,A -85,B 0,C 180,E1 -6198.975,E2 -6198.975} C_VEL
LIN {X 0,Y 495.785,Z 826.182,A -85,B 0,C 180,E1 -6200.001,E2 -6200.001} C_VEL
LIN {X 0,Y 495.544,Z 834.042,A -85,B 0,C 180,E1 -6201.026,E2 -6201.026} C_VEL
LIN {X 0,Y 495.367,Z 841.679,A -85,B 0,C 180,E1 -6202.255,E2 -6202.255} C_VEL
LIN {X 0,Y 495.203,Z 847.799,A -85,B 0,C 180,E1 -6203.482,E2 -6203.482} C_VEL
LIN {X 0,Y 495.173,Z 852.639,A -85,B 0,C 180,E1 -6204.707,E2 -6204.707} C_VEL
LIN {X 0,Y 495.191,Z 856.351,A -85,B 0,C 180,E1 -6205.931,E2 -6205.931} C_VEL
LIN {X 0,Y 495.109,Z 859.708,A -85,B 0,C 180,E1 -6207.56,E2 -6207.56} C_VEL
LIN {X 0,Y 495.046,Z 860.76,A -85,B 0,C 180,E1 -6208.374,E2 -6208.374} C_VEL
LIN {X 0,Y 495.054,Z 861.633,A -85,B 0,C 180,E1 -6210.001,E2 -6210.001} C_VEL
LIN {X 0,Y 495.04,Z 860.807,A -85,B 0,C 180,E1 -6211.628,E2 -6211.628} C_VEL
LIN {X 0,Y 495.098,Z 859.804,A -85,B 0,C 180,E1 -6212.441,E2 -6212.441} C_VEL
LIN {X 0,Y 495.109,Z 858.347,A -85,B 0,C 180,E1 -6213.256,E2 -6213.256} C_VEL
LIN {X 0,Y 495.121,Z 855.33,A -85,B 0,C 180,E1 -6214.478,E2 -6214.478} C_VEL
LIN {X 0,Y 495.251,Z 850.077,A -85,B 0,C 180,E1 -6216.004,E2 -6216.004} C_VEL
LIN {X 0,Y 495.277,Z 843.945,A -85,B 0,C 180,E1 -6217.338,E2 -6217.338} C_VEL
LIN {X 0,Y 495.487,Z 836.831,A -85,B 0,C 180,E1 -6218.566,E2 -6218.566} C_VEL
LIN {X 0,Y 495.66,Z 829.53,A -85,B 0,C 180,E1 -6219.591,E2 -6219.591} C_VEL
LIN {X 0,Y 495.917,Z 820.828,A -85,B 0,C 180,E1 -6220.617,E2 -6220.617} C_VEL
LIN {X 0,Y 496.311,Z 810.168,A -85,B 0,C 180,E1 -6221.642,E2 -6221.642} C_VEL
LIN {X 0,Y 496.641,Z 798.596,A -85,B 0,C 180,E1 -6222.528,E2 -6222.528} C_VEL
LIN {X 0,Y 496.998,Z 787.825,A -85,B 0,C 180,E1 -6223.181,E2 -6223.181} C_VEL
LIN {X 0,Y 497.378,Z 775.755,A -85,B 0,C 180,E1 -6223.743,E2 -6223.743} C_VEL
LIN {X 0,Y 497.726,Z 762.681,A -85,B 0,C 180,E1 -6224.176,E2 -6224.176} C_VEL
LIN {X 0,Y 497.917,Z 748.801,A -85,B 0,C 180,E1 -6224.458,E2 -6224.458} C_VEL
LIN {X 0,Y 498.309,Z 661.857,A -85,B 0,C 180,E1 -6225.741,E2 -6225.741} C_VEL
LIN {X 0,Y 496.399,Z 646.487,A -85,B 0,C 180,E1 -6226.042,E2 -6226.042} C_VEL
LIN {X 0,Y 496.98,Z 621.896,A -85,B 0,C 180,E1 -6229.41,E2 -6229.41} C_VEL
LIN {X 0,Y 497.563,Z 601.796,A -85,B 0,C 180,E1 -6232.2,E2 -6232.2} C_VEL
LIN {X 0,Y 498.314,Z 579.989,A -85,B 0,C 180,E1 -6235.271,E2 -6235.271} C_VEL
LIN {X 0,Y 499.077,Z 558.331,A -85,B 0,C 180,E1 -6238.377,E2 -6238.377} C_VEL
LIN {X 0,Y 498.962,Z 553.076,A -85,B 0,C 180,E1 -6239.157,E2 -6239.157} C_VEL
LIN {X 0,Y 495.778,Z 538.731,A -85,B 0,C 180,E1 -6241.486,E2 -6241.486} C_VEL
LIN {X 0,Y 495.784,Z 538.729,A -85,B 0,C 180,E1 -6244.543,E2 -6244.543} C_VEL
LIN {X 0,Y 495.732,Z 538.733,A -85,B 0,C 180,E1 -6247.562,E2 -6247.562} C_VEL
LIN {X 0,Y 495.769,Z 538.73,A -85,B 0,C 180,E1 -6250.7,E2 -6250.7} C_VEL
LIN {X 0,Y 495.736,Z 538.725,A -85,B 0,C 180,E1 -6254.001,E2 -6254.001} C_VEL
LIN {X 0,Y 495.759,Z 538.732,A -85,B 0,C 180,E1 -6257.12,E2 -6257.12} C_VEL
LIN {X 0,Y 495.761,Z 538.727,A -85,B 0,C 180,E1 -6259.953,E2 -6259.953} C_VEL
LIN {X 0,Y 495.732,Z 538.729,A -85,B 0,C 180,E1 -6262.553,E2 -6262.553} C_VEL
LIN {X 0,Y 495.786,Z 538.729,A -85,B 0,C 180,E1 -6265.457,E2 -6265.457} C_VEL
LIN {X 0,Y 495.756,Z 538.722,A -85,B 0,C 180,E1 -6268.364,E2 -6268.364} C_VEL
LIN {X 0,Y 495.788,Z 538.729,A -85,B 0,C 180,E1 -6271.507,E2 -6271.507} C_VEL
LIN {X 0,Y 495.79,Z 538.72,A -85,B 0,C 180,E1 -6273.932,E2 -6273.932} C_VEL
LIN {X 0,Y 495.76,Z 538.727,A -85,B 0,C 180,E1 -6277.139,E2 -6277.139} C_VEL
LIN {X 0,Y 495.771,Z 538.723,A -85,B 0,C 180,E1 -6280.11,E2 -6280.11} C_VEL
LIN {X 0,Y 495.786,Z 538.715,A -85,B 0,C 180,E1 -6282.681,E2 -6282.681} C_VEL
LIN {X 0,Y 495.794,Z 538.725,A -85,B 0,C 180,E1 -6285.217,E2 -6285.217} C_VEL
LIN {X 0,Y 495.851,Z 538.709,A -85,B 0,C 180,E1 -6288.555,E2 -6288.555} C_VEL
LIN {X 0,Y 495.873,Z 538.717,A -85,B 0,C 180,E1 -6291.852,E2 -6291.852} C_VEL
LIN {X 0,Y 495.895,Z 538.709,A -85,B 0,C 180,E1 -6294.307,E2 -6294.307} C_VEL
LIN {X 0,Y 495.993,Z 538.695,A -85,B 0,C 180,E1 -6297.564,E2 -6297.564} C_VEL
LIN {X 0,Y 496.004,Z 538.696,A -85,B 0,C 180,E1 -6300.812,E2 -6300.812} C_VEL
LIN {X 0,Y 495.844,Z 538.717,A -85,B 0,C 180,E1 -6303.25,E2 -6303.25} C_VEL
LIN {X 0,Y 495.879,Z 538.709,A -85,B 0,C 180,E1 -6306.51,E2 -6306.51} C_VEL
LIN {X 0,Y 495.843,Z 538.716,A -85,B 0,C 180,E1 -6308.97,E2 -6308.97} C_VEL
LIN {X 0,Y 495.828,Z 538.715,A -85,B 0,C 180,E1 -6312.035,E2 -6312.035} C_VEL
LIN {X 0,Y 495.824,Z 538.721,A -85,B 0,C 180,E1 -6315.452,E2 -6315.452} C_VEL
LIN {X 0,Y 495.807,Z 538.718,A -85,B 0,C 180,E1 -6318.247,E2 -6318.247} C_VEL
LIN {X 0,Y 495.774,Z 538.723,A -85,B 0,C 180,E1 -6320.757,E2 -6320.757} C_VEL
LIN {X 0,Y 495.752,Z 538.729,A -85,B 0,C 180,E1 -6323.387,E2 -6323.387} C_VEL
LIN {X 0,Y 495.792,Z 538.725,A -85,B 0,C 180,E1 -6326.068,E2 -6326.068} C_VEL
LIN {X 0,Y 495.772,Z 538.725,A -85,B 0,C 180,E1 -6328.815,E2 -6328.815} C_VEL
LIN {X 0,Y 495.756,Z 538.727,A -85,B 0,C 180,E1 -6331.725,E2 -6331.725} C_VEL
LIN {X 0,Y 495.769,Z 538.725,A -85,B 0,C 180,E1 -6334.694,E2 -6334.694} C_VEL
LIN {X 0,Y 495.73,Z 538.733,A -85,B 0,C 180,E1 -6337.562,E2 -6337.562} C_VEL
LIN {X 0,Y 495.769,Z 538.729,A -85,B 0,C 180,E1 -6340.7,E2 -6340.7} C_VEL
LIN {X 0,Y 495.73,Z 538.733,A -85,B 0,C 180,E1 -6344.002,E2 -6344.002} C_VEL
LIN {X 0,Y 495.72,Z 538.723,A -85,B 0,C 180,E1 -6347.116,E2 -6347.116} C_VEL
LIN {X 0,Y 495.761,Z 538.731,A -85,B 0,C 180,E1 -6349.953,E2 -6349.953} C_VEL
LIN {X 0,Y 495.731,Z 538.733,A -85,B 0,C 180,E1 -6352.553,E2 -6352.553} C_VEL
LIN {X 0,Y 495.785,Z 538.725,A -85,B 0,C 180,E1 -6355.457,E2 -6355.457} C_VEL
LIN {X 0,Y 495.76,Z 538.733,A -85,B 0,C 180,E1 -6358.364,E2 -6358.364} C_VEL
LIN {X 0,Y 495.757,Z 538.733,A -85,B 0,C 180,E1 -6360.759,E2 -6360.759} C_VEL
LIN {X 0,Y 495.114,Z 538.983,A -85,B 0,C 180,E1 -6361.224,E2 -6361.224} C_VEL
LIN {X 0,Y 493.633,Z 539.685,A -85,B 0,C 180,E1 -6361.665,E2 -6361.665} C_VEL
LIN {X 0,Y 490.9,Z 541.81,A -85,B 0,C 180,E1 -6362.358,E2 -6362.358} C_VEL
LIN {X 0,Y 489.956,Z 543.698,A -85,B 0,C 180,E1 -6362.762,E2 -6362.762} C_VEL
LIN {X 0,Y 489.997,Z 545.204,A -85,B 0,C 180,E1 -6363.021,E2 -6363.021} C_VEL
LIN {X 0,Y 491.813,Z 554.135,A -85,B 0,C 180,E1 -6364.39,E2 -6364.39} C_VEL
LIN {X 0,Y 491.335,Z 569.776,A -85,B 0,C 180,E1 -6366.613,E2 -6366.613} C_VEL
LIN {X 0,Y 490.573,Z 592.853,A -85,B 0,C 180,E1 -6369.889,E2 -6369.889} C_VEL
LIN {X 0,Y 490.02,Z 613.241,A -85,B 0,C 180,E1 -6372.686,E2 -6372.686} C_VEL
LIN {X 0,Y 489.893,Z 621.607,A -85,B 0,C 180,E1 -6373.786,E2 -6373.786} C_VEL
LIN {X 0,Y 491.786,Z 634.802,A -85,B 0,C 180,E1 -6374.047,E2 -6374.047} C_VEL
LIN {X 0,Y 491.208,Z 730.62,A -85,B 0,C 180,E1 -6375.473,E2 -6375.473} C_VEL
LIN {X 0,Y 490.935,Z 743.411,A -85,B 0,C 180,E1 -6375.809,E2 -6375.809} C_VEL
LIN {X 0,Y 490.566,Z 756.353,A -85,B 0,C 180,E1 -6376.326,E2 -6376.326} C_VEL
LIN {X 0,Y 490.166,Z 768.94,A -85,B 0,C 180,E1 -6377.022,E2 -6377.022} C_VEL
LIN {X 0,Y 489.837,Z 779.588,A -85,B 0,C 180,E1 -6377.782,E2 -6377.782} C_VEL
LIN {X 0,Y 489.372,Z 790.049,A -85,B 0,C 180,E1 -6378.715,E2 -6378.715} C_VEL
LIN {X 0,Y 489.001,Z 800.339,A -85,B 0,C 180,E1 -6379.859,E2 -6379.859} C_VEL
LIN {X 0,Y 488.629,Z 809.265,A -85,B 0,C 180,E1 -6381.105,E2 -6381.105} C_VEL
LIN {X 0,Y 488.331,Z 816.44,A -85,B 0,C 180,E1 -6382.349,E2 -6382.349} C_VEL
LIN {X 0,Y 488.197,Z 822.411,A -85,B 0,C 180,E1 -6383.645,E2 -6383.645} C_VEL
LIN {X 0,Y 487.972,Z 827.36,A -85,B 0,C 180,E1 -6385.042,E2 -6385.042} C_VEL
LIN {X 0,Y 488.043,Z 829.633,A -85,B 0,C 180,E1 -6385.87,E2 -6385.87} C_VEL
LIN {X 0,Y 487.978,Z 831.492,A -85,B 0,C 180,E1 -6386.697,E2 -6386.697} C_VEL
LIN {X 0,Y 487.933,Z 832.916,A -85,B 0,C 180,E1 -6387.523,E2 -6387.523} C_VEL
LIN {X 0,Y 487.834,Z 834.531,A -85,B 0,C 180,E1 -6389.174,E2 -6389.174} C_VEL
LIN {X 0,Y 487.819,Z 834.769,A -85,B 0,C 180,E1 -6389.999,E2 -6389.999} C_VEL
LIN {X 0,Y 487.893,Z 834,A -85,B 0,C 180,E1 -6391.65,E2 -6391.65} C_VEL
LIN {X 0,Y 487.933,Z 833.039,A -85,B 0,C 180,E1 -6392.476,E2 -6392.476} C_VEL
LIN {X 0,Y 487.978,Z 831.682,A -85,B 0,C 180,E1 -6393.302,E2 -6393.302} C_VEL
LIN {X 0,Y 487.994,Z 828.825,A -85,B 0,C 180,E1 -6394.542,E2 -6394.542} C_VEL
LIN {X 0,Y 488.162,Z 824.939,A -85,B 0,C 180,E1 -6395.783,E2 -6395.783} C_VEL
LIN {X 0,Y 488.252,Z 819.914,A -85,B 0,C 180,E1 -6397.027,E2 -6397.027} C_VEL
LIN {X 0,Y 488.465,Z 813.576,A -85,B 0,C 180,E1 -6398.272,E2 -6398.272} C_VEL
LIN {X 0,Y 488.745,Z 805.693,A -85,B 0,C 180,E1 -6399.518,E2 -6399.518} C_VEL
LIN {X 0,Y 489.051,Z 797.639,A -85,B 0,C 180,E1 -6400.557,E2 -6400.557} C_VEL
LIN {X 0,Y 489.531,Z 787.769,A -85,B 0,C 180,E1 -6401.594,E2 -6401.594} C_VEL
LIN {X 0,Y 489.929,Z 776.588,A -85,B 0,C 180,E1 -6402.538,E2 -6402.538} C_VEL
LIN {X 0,Y 490.296,Z 765.861,A -85,B 0,C 180,E1 -6403.258,E2 -6403.258} C_VEL
LIN {X 0,Y 490.678,Z 753.778,A -85,B 0,C 180,E1 -6403.88,E2 -6403.88} C_VEL
LIN {X 0,Y 491.004,Z 740.49,A -85,B 0,C 180,E1 -6404.373,E2 -6404.373} C_VEL
LIN {X 0,Y 491.168,Z 728.652,A -85,B 0,C 180,E1 -6404.659,E2 -6404.659} C_VEL
LIN {X 0,Y 491.755,Z 635.354,A -85,B 0,C 180,E1 -6406.036,E2 -6406.036} C_VEL
LIN {X 0,Y 489.635,Z 622.251,A -85,B 0,C 180,E1 -6406.312,E2 -6406.312} C_VEL
LIN {X 0,Y 490.08,Z 602.652,A -85,B 0,C 180,E1 -6409.258,E2 -6409.258} C_VEL
LIN {X 0,Y 490.604,Z 584.649,A -85,B 0,C 180,E1 -6412.087,E2 -6412.087} C_VEL
LIN {X 0,Y 491.202,Z 566.67,A -85,B 0,C 180,E1 -6414.965,E2 -6414.965} C_VEL
LIN {X 0,Y 491.589,Z 554,A -85,B 0,C 180,E1 -6416.994,E2 -6416.994} C_VEL
LIN {X 0,Y 489.478,Z 542.955,A -85,B 0,C 180,E1 -6418.854,E2 -6418.854} C_VEL
LIN {X 0,Y 488.749,Z 539.608,A -85,B 0,C 180,E1 -6419.445,E2 -6419.445} C_VEL
LIN {X 0,Y 488.703,Z 539.608,A -85,B 0,C 180,E1 -6422.146,E2 -6422.146} C_VEL
LIN {X 0,Y 488.721,Z 539.613,A -85,B 0,C 180,E1 -6425.113,E2 -6425.113} C_VEL
LIN {X 0,Y 488.678,Z 539.612,A -85,B 0,C 180,E1 -6428.199,E2 -6428.199} C_VEL
LIN {X 0,Y 488.715,Z 539.611,A -85,B 0,C 180,E1 -6431.413,E2 -6431.413} C_VEL
LIN {X 0,Y 488.696,Z 539.603,A -85,B 0,C 180,E1 -6434.023,E2 -6434.023} C_VEL
LIN {X 0,Y 488.74,Z 539.608,A -85,B 0,C 180,E1 -6437.168,E2 -6437.168} C_VEL
LIN {X 0,Y 488.73,Z 539.608,A -85,B 0,C 180,E1 -6439.676,E2 -6439.676} C_VEL
LIN {X 0,Y 488.734,Z 539.633,A -85,B 0,C 180,E1 -6442.267,E2 -6442.267} C_VEL
LIN {X 0,Y 491.604,Z 548.26,A -85,B 0,C 180,E1 -6442.5,E2 -6442.5} C_VEL
LIN {X 0,Y 491.102,Z 619.47,A -85,B 0,C 180,E1 -6443.614,E2 -6443.614} C_VEL
LIN {X 0,Y 491.014,Z 632.216,A -85,B 0,C 180,E1 -6443.972,E2 -6443.972} C_VEL
LIN {X 0,Y 490.881,Z 644.505,A -85,B 0,C 180,E1 -6444.477,E2 -6444.477} C_VEL
LIN {X 0,Y 490.583,Z 656.819,A -85,B 0,C 180,E1 -6445.163,E2 -6445.163} C_VEL
LIN {X 0,Y 490.248,Z 668.46,A -85,B 0,C 180,E1 -6446.007,E2 -6446.007} C_VEL
LIN {X 0,Y 489.927,Z 679.022,A -85,B 0,C 180,E1 -6446.968,E2 -6446.968} C_VEL
LIN {X 0,Y 489.608,Z 687.528,A -85,B 0,C 180,E1 -6447.919,E2 -6447.919} C_VEL
LIN {X 0,Y 489.334,Z 695.867,A -85,B 0,C 180,E1 -6449.06,E2 -6449.06} C_VEL
LIN {X 0,Y 489.033,Z 703.108,A -85,B 0,C 180,E1 -6450.277,E2 -6450.277} C_VEL
LIN {X 0,Y 488.792,Z 709.727,A -85,B 0,C 180,E1 -6451.674,E2 -6451.674} C_VEL
LIN {X 0,Y 488.667,Z 714.764,A -85,B 0,C 180,E1 -6453.082,E2 -6453.082} C_VEL
LIN {X 0,Y 488.524,Z 718.328,A -85,B 0,C 180,E1 -6454.432,E2 -6454.432} C_VEL
LIN {X 0,Y 488.471,Z 720.096,A -85,B 0,C 180,E1 -6455.339,E2 -6455.339} C_VEL
LIN {X 0,Y 488.416,Z 721.325,A -85,B 0,C 180,E1 -6456.24,E2 -6456.24} C_VEL
LIN {X 0,Y 488.407,Z 722.08,A -85,B 0,C 180,E1 -6457.137,E2 -6457.137} C_VEL
LIN {X 0,Y 488.42,Z 722.396,A -85,B 0,C 180,E1 -6458.03,E2 -6458.03} C_VEL
LIN {X 0,Y 488.447,Z 722.03,A -85,B 0,C 180,E1 -6459.264,E2 -6459.264} C_VEL
LIN {X 0,Y 488.514,Z 720.531,A -85,B 0,C 180,E1 -6460.677,E2 -6460.677} C_VEL
LIN {X 0,Y 488.609,Z 718.711,A -85,B 0,C 180,E1 -6461.676,E2 -6461.676} C_VEL
LIN {X 0,Y 488.728,Z 715.78,A -85,B 0,C 180,E1 -6462.855,E2 -6462.855} C_VEL
LIN {X 0,Y 488.927,Z 710.603,A -85,B 0,C 180,E1 -6464.376,E2 -6464.376} C_VEL
LIN {X 0,Y 489.15,Z 704.847,A -85,B 0,C 180,E1 -6465.65,E2 -6465.65} C_VEL
LIN {X 0,Y 489.451,Z 697.4,A -85,B 0,C 180,E1 -6466.95,E2 -6466.95} C_VEL
LIN {X 0,Y 489.789,Z 688.4,A -85,B 0,C 180,E1 -6468.205,E2 -6468.205} C_VEL
LIN {X 0,Y 490.131,Z 678.921,A -85,B 0,C 180,E1 -6469.257,E2 -6469.257} C_VEL
LIN {X 0,Y 490.494,Z 668.353,A -85,B 0,C 180,E1 -6470.203,E2 -6470.203} C_VEL
LIN {X 0,Y 490.776,Z 658.162,A -85,B 0,C 180,E1 -6470.937,E2 -6470.937} C_VEL
LIN {X 0,Y 491.01,Z 645.945,A -85,B 0,C 180,E1 -6471.619,E2 -6471.619} C_VEL
LIN {X 0,Y 491.143,Z 632.656,A -85,B 0,C 180,E1 -6472.161,E2 -6472.161} C_VEL
LIN {X 0,Y 491.201,Z 620.118,A -85,B 0,C 180,E1 -6472.498,E2 -6472.498} C_VEL
